(* CODESYS project devicelib.library
   Author: AMKO-Engineering
   Placeholder: Device_Library
   Title: Device_Library
   Version: 1.2.0.0
   Description: Device library of AMKO-Engineering.
   Company: AMKO-Engineering

Project tree, tasks and I/O mapping:
  libraries: System_Library, * (AMKO-Engineering); Tc2_MC2, 3.3.38.0 (Beckhoff Automation GmbH); Tc2_MC2_Drive, 3.3.21.0 (Beckhoff Automation GmbH); Tc2_Standard, 3.3.3.0 (Beckhoff Automation GmbH); Utilities_Library, * (AMKO-Engineering)
  Actuators/
    Cylinder/
      DataTypes/
        data type E_CylinderCmd
        data type E_ValveResetState
      Functions/
        function block Fb_DevCylWithFbk [ST]: ExecCalcTimers, ExecDirection, ExecSetFeedback, ExecTimeout, CmdSimulate, CmdTeach, Init
        function block FB_DevValve [ST]: ExecSetFeedback, ExecSetOutPuts, CmdClose, CmdHold, CmdManual, CmdOpen, CmdReset, CmdSafeStop, CmdTeach, Init
      MLTFunctions/
        function block Fb_DevSupportCyl [ST]: ExecCalc, ExecCylControl, ExecFaultHandling, Init_Support, Mod_ManualControl, Mod_SupportDown
  Axis/
    DataTypes/
      data type E_AxisCmd
      data type UDT_AxisData
      data type UDT_AxVal
    FunctionBlocks/
      function block FB_Axis [ST]: GearAsSlave, GearOutSlave, GearSlaveDyn, GetActVal, Hold, Home, Init, Jog, MoveAbs, MoveModulo, MoveRelative, MoveVeloFwd, MoveVeloRev, Reset, Stop
      function block Fb_AxisNew [ST]: CmdGearDynamic, CmdGearIn, CmdGearOut, CmdHalt, CmdHome, CmdJog, CmdLimitVelocity, CmdMoveAbs, CmdMoveModulo, CmdMoveRelative, CmdMoveVelocity, CmdReset, CmdSafeSpeed, CmdSafeStop, Init, ExecGearDynamic, ExecGearIn, ExecGearOut, ExecHalt, ExecHome, ExecJog, ExecMoveAbsolute, ExecMoveModulo, ExecMoveRelative, ExecMoveVelocity, ExecEnable, ExecReadStatus, ExecReset, ExecSafeFunctions, METH_ExecuteMotionFunctions, METH_ExecuteOrganizationFunctions
    Interface/
  BaseFunctions/
    function block FB_DevBase [ST]: CmdReset, CmdSafeStop
  Buttons/
    DataTypes/
    Functions/
      function block FB_DevHMIButton [ST]
      function block FB_DevPushButton [ST]
      function block FB_DevPushbuttonLight [ST]
  Encoders/
    DataTypes/
    FunctionBlocks/
      function block FB_EncoderBase [ST]: FastTask
      function block FB_EncoderInput [ST]: FastTask
  GroupHandlers/
    ManualControlHandler/
      function block FB_DevManualHandler [CFC]
  Heaters/
    function block FB_DevPWMGenerator [ST]: CalcCycle, ExecSetOutput, CmdOutputCycle, CmdOutputOff, CmdOutputOn
  Lights/
    DataTypes/
      data type E_LightState
    Functions/
      function block Fb_DevLight [ST]: Mod_SetOutput
  Outputs/
    DigitalOutputs/
      function block FB_DigitalOutput [ST]: ExecSetFeedback, ExecSetOutput, CmdOn
  Sensors/
    DigitalSensor/
      DataTypes/
        data type Udt_DigitalSensor
      FunctionBlocks/
        function block Fb_DevDigitalInput [ST]
        function block Fb_DevDigitalInputFunctions [ST]
    FootPedals/
      DataTypes/
        data type E_FootpedalPos
      FunctionBlocks/
        function block FB_EfkaEB301A_FootPedal [ST]: ACT_ConvertGreycode, ACT_CreateEdges
  Version/
    global variables Global_Version
*)

// Actuators/Cylinder/DataTypes/E_CylinderCmd
(* cylinder commands *)
TYPE E_CylinderCmd :
(
	Cyl_Idle 		:= 0,// Jog Cylinder command Referance 0 Idle (wait for command)
	Cyl_Init 		:= 1,// Jog Cylinder command Referance 1 initialize Cylinder
	Cyl_Enable 		:= 2,// Jog Cylinder command Referance 2 enable
	Cyl_Disable 	:= 3,// Jog Cylinder command Referance 3 disable
	Cyl_Reset 		:= 4,// Jog Cylinder command Referance 4 reset
	Cyl_Hold 		:= 5,// Jog Cylinder command Referance 5 hold
	Cyl_Teach 		:= 6,// Jog Cylinder command Referance 6 teach timeout settings
	Cyl_Calculate 	:= 7,// Jog Cylinder command Referance 7 calculate timeout settings from parameters
	Cyl_Expand 		:= 8,// Jog Cylinder command Referance 8 expand
	Cyl_Retract 	:= 9 // Jog Cylinder command Referance 9 retract
);
END_TYPE

// Actuators/Cylinder/DataTypes/E_ValveResetState
{attribute 'qualified_only'}
{attribute 'strict'}
TYPE E_ValveResetState :
(
	Res_Idle 		:= 0,
	Res_Closed		:= 1,
	Res_Open		:= 2
);
END_TYPE

// Axis/DataTypes/E_AxisCmd
(* axis command structure *)
TYPE E_AxisCmd :
(
	Ax_Idle 		:= 0,// Axis command Referance 0 Axis Idle
	Ax_Init 		:= 1,// Axis command Referance 1 Initialize axis
	Ax_Enable 		:= 2,// Axis command Referance 2 Enable
	Ax_Disable 		:= 3,// Axis command Referance 3 Disable
	Ax_Reset 		:= 4,// Axis command Referance 4 Reset
	Ax_Hold 		:= 5,// Axis command Referance 5 Hold
	Ax_Home 		:= 6,// Axis command Referance 6 Home
	Ax_JogFwd 		:= 7,// Axis command Referance 7 Jog Forward
	Ax_JogRev 		:= 8,// Axis command Referance 8 Jog Reverse
	Ax_MoveRelative := 9,// Axis command Referance 9 Move axis relative
	Ax_MoveAbs 		:= 10,// Axis command Referance 11 Move absolute reverse
	Ax_MoveModulo 	:= 11,// Axis command Referance 11 Move Module
	Ax_MoveVeloFwd 	:= 12,// Axis command Referance 12 Move velocity forward
	Ax_MoveVeloRev 	:= 13,// Axis command Referance 13 Move velocity reverse
	Ax_HardStop 	:= 14,// Axis command Referance 14 hard stop or emergency stop
	Ax_SoftStop 	:= 15,// Axis command Referance 15 soft stop after motion command
	Ax_GearSlave 	:= 16,// Axis command Referance 16 gear axis as slave
	Ax_GearSlaveDyn	:= 17,// Axis command Referance 17 gear axis as slave dynamic
	Ax_GearOutSlave := 18,// Axis command Referance 18 gear out from Master axis 
	Ax_Maintenance	:= 50 // Axis Command referance 50 maintenance mode, axis enabled with no command active
);
END_TYPE

// Axis/DataTypes/UDT_AxisData
TYPE UDT_AxisData:
STRUCT
	// ===== Axis name =====
		AxisName	: STRING 	; // Name of the axis (used for fault handling and identification)
		AxisNumber	: INT		; // Axis number 

	// ===== Fault data =====
		Message			: UDT_Fault 	; // Message data from Cylinder
		MessageActive	: BOOL			; // Message is active
		ErrorActive 	: BOOL 			;	// Axis in error state

	// ===== Axis Commands =====
		// ***** Enable command	*****
			CmdEnable		: BOOL 		; // Command enable axis
		// ***** Active commands *****
			AxisCmd			: E_AxisCmd ; // Axis command
			AxisSafeCmd		: E_AxisCmd	; // Axis safe command
			AxisAct			: E_AxisCmd ; // Axis Active status
		// ***** Command Modes *****
			CmdHomingMode 	: MC_HomingMode ; // Homing Mode ( MC_DefaultHoming, MC_Direct, MC_ForceCallibration, MC_ResetCallibration)
			CmdJogMode		: E_JogMode 	;
			CmdBuffermode	: MC_BufferMode	; // Buffermode used for command transition 	 
	// ===== Axis Safe commands =====
		SafeCmdLimitVelo: BOOL 	; // safe command limit velocity
		SafeCmdVelocity	: LREAL ; // Safe command velocity
		SafeCmdStop		: BOOL 	; // Stop command from safety or collision detection		
		SafeVeloLimit	: LREAL ; // safe velocity limit (link to FPAR)
	// ===== Status indication active =====
		ActHoming	: BOOL ; // Axis is homing
		ActBusy		: BOOL ; // Axis is Busy 
		ActMoving	: BOOL ; // Axis is moving
		ActAtVelo	: BOOL ; // Axis is at command velocity (only when written in Move velocity mode)

	// ===== Status indication done  =====
		FcoInit		: BOOL ; // Axis is initialised
		FcoIdle		: BOOL ; // Axis is idle enable required
		FcoEnabled	: BOOL ; // Axis is enabled
		FcoHomed	: BOOL ; // Axis is homed
		FcoGeared	: BOOL ; // Axis is geared to master axis
		FcoHeld		: BOOL ; // Axis is holding
		FcoStopped	: BOOL ; // Axis is stopped
		FcoReset	: BOOL ; // Axis reset done
		FcoReady 	: BOOL ; // Axis is ready for command
		FcoAtCmdPos	: BOOL ; // Axis is at command position (tol 0.2 deg)
		FcoCmdActive: BOOL ; // Axis new command values are active
		
	// ===== Move values =====
		Pos			: UDT_Axval	; // possition values (0 = infinite)
		Velocity 	: UDT_AxVal	; // Velocity values
		Accel		: UDT_Axval ; // Aceleration values
		Decel		: UDT_Axval ; // Deceleration values
		Torque		: UDT_Axval ; // Torque values
		EncTurnoverVal	: DINT 	; // Encoder turnover value
		TimeDisableDelay : TIME ; // Time off delay after axis move command (remove enable)
		
	// ===== Config Bits =====
		IcfCommandSpeedRpm	: BOOL ; // input speeds in Rpm
		IcfEnableForward 	: BOOL ; // Enable forward motion
 		IcfEnablereverse	: BOOL ; // Enable reverse motion
		IcfContinuous		: BOOL ; // continuous motion possible (no endpoint)
		IcfAlwaysEnable		: BOOL ; // 1 = Axis always enabled, 0 = Axis disabled at Idle 
		
	// ===== Master Axis =====
		MasterAxisRef	: REFERENCE TO AXIS_REF ; // Master axis reference (if applicable)
		GearMasterRev	: UINT	:= 1	; // Master Axis Gearing revolutions (Denominator)
		GearSlaveRev	: LREAL	:= 1	; // Slave Axis gearing revolutions (numerator)	
		ReverseSlave	: BOOL 	; // Reverse slave axis relative to master
		 
END_STRUCT
END_TYPE

// Axis/DataTypes/UDT_AxVal
TYPE UDT_AxVal :
STRUCT
	// ***** Velocity settings *****
		HardMax		: LREAL 	; // Hardware maximum set absolute maximum
		ManMax 		: LREAL		; // Manual maximum percentage of hardware max
		AutoMax		: LREAL		; // Automatic maximum percentage of hardware max
		HomeMax		: LREAL 	; // Homing maximum percentage of hardware max
		CmdVal		: LREAL 	; // Commanded value
		SafeVal		: LREAL		; // Command value after safety check
		PrevVal		: LREAL		; // previous command value 
		ActVal		: LREAL		; // Actual value
		ActModulo	: LREAL		; // [deg] Modulo position
		RefVal		: LREAL 	; // referance value (basic setting or home) 
END_STRUCT
END_TYPE

// Lights/DataTypes/E_LightState
(* discribes signal light state *)
TYPE E_LightState :
(
	Light_Off 		:= 0,// Jog Light state Referance 0 Light is off
	Light_BlinkSlow := 1,// Jog Light state Referance 1 Light blinking fast 
	Light_BlinkFast := 2,// Jog Light state Referance 2 light blinking slow
	Light_On 		:= 3 // Jog Light state Referance 3 Light permanently on
);
END_TYPE

// Sensors/DigitalSensor/DataTypes/Udt_DigitalSensor
TYPE Udt_DigitalSensor :
STRUCT
	Istatus		AT 	%I* : BOOL			;// Digital sensor, Direct input status
	ISensorEnable		: BOOL			;// Digital sensor, Input enable button
	tSensorDelay		: TIME 			;// Time before delayed signal becomes active 
	FcoSensorActive		: BOOL 			;// Digital sensor, Button active state
	FcoDelay			: BOOL			;// Digital sensor, Delayed input status (3 seconds) 
	FeStatus			: BOOL			;// Digital sensor, Falling edge of input signal	
	ReStatus			: BOOL			;// Digital sensor, Rising edge of input signal
	FcoFlipFlop			: BOOL			;// Digital sensor, feedback flip flop
	TetSensorActive		: TIME			;// Digital sensor, Time elapsed while button is active
END_STRUCT
END_TYPE

// Sensors/FootPedals/DataTypes/E_FootpedalPos
{attribute 'qualified_only'}
{attribute 'strict'}
TYPE E_FootpedalPos :
(
	eReverse2 	,
	eReverse1 	,
	eIdle		,
	eForward1	,
	eForward2	,
	eForward3	,
	eForward4	,
	eForward5	,
	eForward6	,
	eForward7	,
	eForward8	,
	eForward9	,
	eForward10	,
	eForward11	,
	eForward12	,
	eForward13	,
	eFalse			
) INT; 
END_TYPE

// Version/Global_Version
{attribute 'TcGenerated'}
{attribute 'no-analysis'}
{attribute 'linkalways'}
// This function has been automatically generated from the project information.
VAR_GLOBAL CONSTANT
	{attribute 'const_non_replaced'}
	stLibVersion_Device_Library : ST_LibVersion := (iMajor := 1, iMinor := 2, iBuild := 0, iRevision := 0, nFlags := 0, sVersion := '1.2.0.0');
END_VAR

// Actuators/Cylinder/Functions/Fb_DevCylWithFbk
FUNCTION_BLOCK PUBLIC Fb_DevCylWithFbk EXTENDS FB_DevValve
VAR_INPUT
	bIcfFbkOpenPresent 	: BOOL := FALSE ; // Feedback for cylinder open is present 
	bIcfFbkClosedPresent: BOOL := FALSE ; // Feedback for Cylinder closed is present
	bIcfTimeChecked		: BOOL := TRUE 	; // Cylinder timing is checked = default true
	nMargin				: LREAL:= 10	; // % of tollerance in move speed 
END_VAR
VAR_OUTPUT
	// ===== Teach function =======
	bCmdCopyTimeParam 	: BOOL	:= FALSE 	;// Cylinder, Command to higher level copy toucht time to parameters
	nOutTimeToClose		: LREAL	:= 0		; // Time it takes for valve to open	
	nOutTimeToOpen		: LREAL := 0		; // Time it takes for valve to close
	bFeClosed			: BOOL 	:= FALSE	; // closed sensor falling edge
	bReClosed			: BOOL 	:= FALSE	; // closed sensor rising edge
	bFeOpen				: BOOL 	:= FALSE 	; // Open sensor falling edge
	bReOpen				: BOOL 	:= false 	; // open sensor rising edge 
END_VAR
VAR	
	bFcoCalcDone	: BOOL := FALSE ; // Calculate timers done 
	
	stTimesClose	: Udt_TimerBandwith ; // Timer bandwith for cylinder close
	stTimesOpen		: Udt_TimerBandwith	; // Timer bandwitch for cylinder open 
	
	fbSensorClosed	: Fb_DevDigitalInputFunctions ; // Digital sensor function closed detection
	fbSensorOpen	: Fb_DevDigitalInputFunctions ; // Digital sensor function open detection
	
	fbTimerOpen		: TON ; // Timer for cylinder to open
	fbTimerClose 	: TON ; // Timer for cylinder to close
	fbTimerTeach	: TON ; // timer for teachin cylinder 

	rtCmdWriteParam	: R_TRIG ; // Write parameter rising edge trigger 
	// Simulation
	fbTimerSimOpen 	: TON 	; 
	fbTimerSimClose	: TON 	; 
	
	// Time Cylinder valid 
	bTriggerTimeClose	: BOOL ;
	bTriggerTimeOpen	: BOOL ;

END_VAR

IF NOT bInitOk THEN
	RETURN;
ELSE
	SUPER^();
END_IF 

// ====== Check direction of movement =======
	ExecDirection();
	
// ====== Check movement speed =======
	IF bFcoCalcDone AND bIcfTimeChecked THEN 
		ExecTimeout();
	END_IF
	
// ====== Calculate timers =======
	IF nTimeToCloseMs <> stTimesClose.Nominal OR nTimeToOpenMs <> stTimesOpen.Nominal OR NOT bFcoCalcDone THEN 
		bFcoCalcDone := FALSE ;
		ExecCalcTimers();
	END_IF

// ==== set timer output feedback 
	nOutTimeToClose := stTimesClose.Nominal ;
	nOutTimeToOpen	:= stTimesOpen.Nominal	;	

// ===== send write parameters command ======	
	rtCmdWriteParam(CLK := bFcoCalcDone);
	bCmdCopyTimeParam := rtCmdWriteParam.Q	;

METHOD PRIVATE ExecCalcTimers : BOOL
VAR
END_VAR
// ====== Calculate close times ======
	stTimesClose.Nominal 	:= nTimeToCloseMs ;
	stTimesClose.Maximum 	:= nTimeToCloseMs * (1 + (nMargin / 100));
	stTimesClose.Minimal 	:= nTimeToCloseMs * (1 - (nMargin / 100));

// ====== Calculate open times ======
	stTimesOpen.Nominal 	:= nTimeToOpenMs ;
	stTimesOpen.Maximum 	:= nTimeToOpenMs * (1 + (nMargin / 100));
	stTimesOpen.Minimal 	:= nTimeToOpenMs * (1 - (nMargin / 100));
	
// ====== Set feedback =======
	bFcoCalcDone := TRUE ;
END_METHOD

METHOD PRIVATE ExecDirection : BOOL
VAR_INPUT
END_VAR
// ===== Check direction commands =====
 	IF q_Close AND fbSensorOpen.bReStatus AND NOT q_Open THEN
		stFault.MessageNumber	:= E_MessageNumbers.CF_WrongDirection 	;
		stFault.Discription		:= 'Cylinder Opening instead of closing';
		stFault.FaultType		:= E_FaultTypes.CF 					;
		bErrorActive			:= TRUE 								;
		refFbFault.CmdAddFault( stFault );
	ELSIF q_Open AND fbSensorClosed.bReStatus AND NOT q_close THEN
		stFault.MessageNumber	:= E_MessageNumbers.CF_WrongDirection 	;
		stFault.Discription		:= 'Cylinder closing instead of opening';
		stFault.FaultType		:= E_FaultTypes.CF 					;
		bErrorActive			:= TRUE 								;
		refFbFault.CmdAddFault( stFault );
	END_IF
END_METHOD

METHOD PROTECTED ExecSetFeedback : BOOL
VAR_INPUT
END_VAR
// ====== Call sensor Open function =======
	IF bIcfFbkClosedPresent THEN 
		fbSensorClosed();
		bFco_Closed := fbSensorClosed.bFcoInputActive ;
		bFeClosed 	:= fbSensorClosed.bFeStatus ;
		bReClosed 	:= fbSensorClosed.bReStatus ;
	ELSE 
		fbTOnClose	(IN 	:= q_Close, PT 	:= LREAL_TO_TIME(nTimeToCloseMs))	;
		bFco_Closed := fbTOnClose.Q ;
	END_IF

// ====== Call sensor Close function =======
	IF bIcfFbkOpenPresent THEN 
		fbSensorOpen() 	;
		bFco_open 	:= fbSensorOpen.bFcoInputActive ;
		bFeOpen		:= fbSensorOpen.bFeStatus;
		bReOpen		:= fbSensorOpen.bReStatus;
	ELSE 
		FbTOnOpen	(IN 	:= q_Open, PT 	:= LREAL_TO_TIME(nTimeToOpenMs))	;
		bFco_Open := FbTOnOpen.Q ;
	END_IF

// ====== set outputs =======
	bReady		:= bFco_Closed OR bFco_Open ;
END_METHOD

METHOD PRIVATE ExecTimeout : BOOL
VAR_INPUT
END_VAR
VAR
	nTimePassedMs : LREAL ;
END_VAR
// ====== Set triggers ======
	IF q_Close  AND bFco_Open THEN 
		bTriggerTimeClose := TRUE ;
	ELSIF q_Open OR bFco_Closed  THEN 
		bTriggerTimeClose := FALSE ;
	END_IF

	IF q_Open  AND bFco_Closed THEN 
		bTriggerTimeOpen := TRUE ;
	ELSIF q_Close OR bFco_Open THEN
		bTriggerTimeOpen := FALSE ;
	END_IF
	
//======= run timers =======
	IF bIcfFbkClosedPresent THEN 
		fbTimerClose(IN := q_Close, PT := T#1M);
	END_IF	
	
	IF bIcfFbkOpenPresent THEN 
		fbTimerOpen	(IN := q_Open , PT := T#1M);
	END_IF

//====== Run timeout checks for cylinder close =======
	nTimePassedMs:= TIME_TO_LREAL(fbTimerClose.ET);
	
	IF bIcfFbkClosedPresent THEN 
		IF bTriggerTimeClose THEN 
			IF fbSensorClosed.bReStatus THEN 
				IF nTimePassedMs < stTimesClose.Minimal THEN 
					// send message to HMI 
					stFault.MessageNumber	:= E_MessageNumbers.CF_MoveToFast 	;
					stFault.Discription		:= 'Cylinder closing to fast'		;
					stFault.FaultType		:= E_FaultTypes.CF 				;
					bErrorActive			:= TRUE 							;
					refFbFault.CmdAddFault( stFault );
				ELSIF	nTimePassedMs > stTimesClose.Maximum  THEN
					// send message to HMI 
					stFault.MessageNumber	:= E_MessageNumbers.CF_MoveToSlow 	;
					stFault.Discription		:= 'Cylinder closing to Slow'		;
					stFault.FaultType		:= E_FaultTypes.CF 				;
					bErrorActive			:= TRUE 							;
					refFbFault.CmdAddFault( stFault );
				END_IF
			END_IF
		END_IF
	END_IF	

//====== Run timeout checks for cylinder Open =======
	nTimePassedMs:= TIME_TO_REAL(fbTimerOpen.ET);

	IF bIcfFbkOpenPresent THEN 
		IF bTriggerTimeOpen THEN 
			IF fbSensorOpen.bReStatus THEN 
				IF nTimePassedMs < stTimesOpen.Minimal THEN 
					// send message to HMI 
					stFault.MessageNumber	:= E_MessageNumbers.CF_MoveToFast 	;
					stFault.Discription		:= 'Cylinder Opening to fast'		;
					stFault.FaultType		:= E_FaultTypes.CF 				;
					bErrorActive			:= TRUE 							;
					refFbFault.CmdAddFault( stFault );
				ELSIF	nTimePassedMs > stTimesOpen.Maximum  THEN
					// send message to HMI 
					stFault.MessageNumber	:= E_MessageNumbers.CF_MoveToSlow 	;
					stFault.Discription		:= 'Cylinder Opening to Slow'		;
					stFault.FaultType		:= E_FaultTypes.CF 				;
					bErrorActive			:= TRUE 							;
					refFbFault.CmdAddFault( stFault );
				END_IF
			END_IF
		END_IF
	END_IF
END_METHOD

METHOD PUBLIC CmdSimulate : BOOL
VAR_INPUT
	bFbkReverse		: BOOL := FALSE ; 
	tTimeSimOpen	: TIME := T#1S 	;
	tTimeSimClose	: TIME := T#1S 	;  
END_VAR
VAR
	bCmdSimulate : BOOL := TRUE ;
END_VAR
// Run timers when cylinder is active 
	fbTimerSimOpen	(IN := q_Open	, PT := tTimeSimOpen);
	fbTimerSimClose	(IN := q_Close	, PT := tTimeSimClose);

 // set feedback sensors to simulate
	fbSensorOpen.bCmdSimulate 	:= TRUE ;
	fbSensorClosed.bCmdSimulate := TRUE ;

 // set simulated feedback state 
	IF bFbkReverse THEN 
		fbSensorClosed.bSimState:= fbTimerSimOpen.Q 	;
		fbSensorOpen.bSimState	:= fbTimerSimClose.Q 	; 	
	ELSE 
		fbSensorClosed.bSimState:= fbTimerSimClose.Q 	;
		fbSensorOpen.bSimState	:= fbTimerSimOpen.Q 	; 	
	END_IF
END_METHOD

METHOD PUBLIC CmdTeach : BOOL
VAR_INPUT
END_VAR
// ====== turn off time check function until new calculation cycle =======
	bFcoCalcDone := false ;

// ====== teach cylinder from hardware inputs ======
	fbTimerTeach	(PT:= T#60S);
	fbTimerSwitchDir(PT:= T#1S); 
// ====== time cylinder cycles ======
	// ===== Start test loop =====
	IF bFco_Closed AND fbTimerSwitchDir.Q THEN
		bCmdClose 			:= FALSE;
		bCmdOpen 			:= TRUE ;
		fbTimerSwitchDir.IN	:= FALSE; 
		fbTimerTeach.IN 	:= TRUE ;
	ELSIF bFco_Open AND fbTimerSwitchDir.Q THEN
		bCmdClose 			:= TRUE ;
		bCmdOpen 			:= FALSE;
		fbTimerSwitchDir.IN	:= FALSE; 
		fbTimerTeach.IN 	:= TRUE ;
	ELSIF NOT bCmdClose AND NOT bCmdOpen THEN 
		bCmdClose 			:= TRUE ;
		bCmdOpen 			:= FALSE;
		fbTimerTeach.IN 	:= TRUE ;
	END_IF

// ====== start timing ========
	IF bCmdClose AND bFco_Closed THEN 
		IF fbTimerTeach.IN THEN
			nTimeToCloseMs 	:= TIME_TO_LREAL(fbTimerTeach.ET);
		END_IF
		fbTimerSwitchDir.IN := TRUE 		;
		fbTimerTeach.IN 	:= FALSE 		;
	ELSIF bCmdOpen AND bFco_Open THEN 
		IF fbTimerTeach.IN THEN
			nTimeToOpenMs		:= TIME_TO_LREAL(fbTimerTeach.ET);
		END_IF
		fbTimerSwitchDir.IN := TRUE 		;
		fbTimerTeach.IN 	:= FALSE 		;
	END_IF
END_METHOD

METHOD PUBLIC Init : BOOL
VAR_INPUT
	// Valve data
	nInValveNumber	: UDINT				:= 0		; // Cylinder identification number
	// Command state
	eResetState		: E_ValveResetState := 0		; // Cylinder reset state variable (default is idle) 
	eSafeState		: E_ValveResetState	:= 0		; // Valve safe state
END_VAR
bFcoCalcDone := FALSE;

// Enable sensor feedback
fbSensorClosed.bEnable	:= TRUE ;
fbSensorOpen.bEnable	:= TRUE ;

// Call feedback sensors 
ExecSetFeedback(); 

SUPER^.Init(nInValveNumber, eResetState, eSafeState);
END_METHOD

END_FUNCTION_BLOCK

// Actuators/Cylinder/Functions/FB_DevValve
FUNCTION_BLOCK PUBLIC FB_DevValve EXTENDS FB_DevBase
VAR_INPUT
	// Timer values
	nTimeToCloseMs	: LREAL			:= 50		; // Time it takes for valve to open	
	nTimeToOpenMs	: LREAL			:= 50		; // Time it takes for valve to close
END_VAR
VAR_OUTPUT
	// ===== Status indicators =======
		bFco_Closed		:	BOOL := FALSE ;
		bFco_Open		: 	BOOL := FALSE ;
END_VAR
VAR
	// Hardware links 
		q_Open			AT %Q* : BOOL := FALSE 	; // Open valve
		q_Close 		AT %Q* : BOOL := FALSE	; // Close valve
	// Internal commands
		bCmdClose 	: BOOL := FALSE ; // close valve 
		bCmdOpen	: BOOL := FALSE ; // Open valve
		bCmdHold	: BOOL := FALSE ; // Hold valve status change
	// Time functions 
		fbTOnClose	: TON	; // Timer for valve close
		FbTOnOpen	: TON 	; // Timer for valve Open
		fbTimerSwitchDir: TON ; // Time for teach function switch direction 
	// reset and safe state
		eResetState		: E_ValveResetState := 0		; // Cylinder reset state variable (default is idle) 
		eSafeState		: E_ValveResetState	:= 0		; // Valve safe state
END_VAR

// ===== hold all actions if not initialized ======
IF NOT bInitOk THEN
	RETURN;
ELSE
	SUPER^();
END_IF 


// ====== Set Outputs =======
	ExecSetOutPuts();

// ===== collect feedback ======
	ExecSetFeedback();

// ===== Message test function ======
	IF bMessageTest THEN 
		stFault.Active 			:= TRUE ;
		stFault.Discription 	:= 'This is a test message from fb_DevValve';
		stFault.MessageNumber 	:= E_MessageNumbers.OM_MessageTest ;
		stFault.FaultType		:= Utilities_Library.E_FaultTypes.OM ;
		refFbFault.CmdAddFault( stFault );
	END_IF

METHOD PROTECTED ExecSetFeedback : BOOL
VAR_INPUT
END_VAR
// ====== Set timers =======
	fbTOnClose	(PT 	:= LREAL_TO_TIME(nTimeToCloseMs))	;
	FbTOnOpen	(PT		:= LREAL_TO_TIME(nTimeToOpenMs))	;

// ====== Set timed feedback ======
	IF q_Close THEN 
		fbTOnClose.IN 	:= TRUE ;
		fbTOnopen.IN 	:= FALSE;
	ELSIF q_Open THEN 
		fbTOnClose.IN 	:= FALSE;
		FbTOnOpen.IN	:= TRUE ;
	ELSE 
		fbTOnClose.IN 	:= FALSE;
		FbTOnOpen.IN	:= FALSE;
	END_IF
	
// ====== set outputs =======
	bFco_Closed := fbTOnClose.Q ;
	bFco_Open	:= FbTOnOpen.Q	;
	bReady		:= bFco_Closed OR bFco_Open ;
END_METHOD

METHOD PROTECTED ExecSetOutPuts : BOOL
VAR_INPUT
END_VAR
// ======= Set Outputs according to commands and check safety features =======
	IF bEnable	OR bCmdManual THEN  
		IF NOT bCmdHold THEN 
			q_Close	:= bCmdClose;
			q_Open	:= bCmdOpen	;
		END_IF
	ELSE
		CASE eSafeState OF 
			E_ValveResetState.Res_Idle:
				q_Close	:= bFco_Closed;		
				q_Open 	:= bFco_Open;
			E_ValveResetState.Res_Closed:
				q_Close	:= TRUE	;		
				q_Open 	:= FALSE;
			E_ValveResetState.Res_Open:
				q_Close	:= FALSE;		
				q_Open 	:= TRUE	;
		END_CASE
		bCmdClose 	:= bFco_Closed 	;
		bCmdOpen	:= bFco_Open	;
		bCmdHold	:= FALSE ; 
	END_IF
END_METHOD

METHOD PUBLIC CmdClose : BOOL // close valve or retract cylinder
VAR_INPUT
END_VAR
// ====== Set close command if enabled ======
	bCmdClose 	:= TRUE	;		
	bCmdOpen 	:= FALSE;
	
// ===== Set feedback ======
	CmdClose := bFco_Closed ;
END_METHOD

METHOD PUBLIC CmdHold : BOOL
VAR_INPUT
END_VAR
// ====== set hold command =====
	bCmdHold := TRUE ;
END_METHOD

METHOD PUBLIC CmdManual : BOOL
VAR_INPUT
	bCmdOpen	: BOOL ; // open valve 
	bCmdClose	: BOOL ; // Close valve
	bCmdTeach	: BOOL ; // Teach valve  
END_VAR
// Enable manual commands
bCmdManual S= TRUE ;

// execute manual command 
	IF bCmdOpen THEN 
		CmdOpen();
	ELSIF bCmdClose THEN 
	 	CmdClose(); 
	ELSIF bCmdTeach THEN
		CmdTeach ();
	END_IF
END_METHOD

METHOD PUBLIC CmdOpen : BOOL // Open valve or retract cylinder
VAR_INPUT
END_VAR
// ====== Set open command if enabled ======
	bCmdClose 	:= FALSE;		
	bCmdOpen 	:= TRUE	;
	
// ===== Set feedback ======
	CmdOpen := bFco_Open ;
END_METHOD

METHOD CmdReset : BOOL
VAR_INPUT
END_VAR
// ====== Set outputs according to reset state =======
	IF bEnable THEN 
		CASE eResetState OF 
			E_ValveResetState.Res_Idle:
				bCmdClose 	:= FALSE;		
				bCmdOpen 	:= FALSE;
			E_ValveResetState.Res_Closed:
				bCmdClose 	:= TRUE	;		
				bCmdOpen 	:= FALSE;
			E_ValveResetState.Res_Open:
				bCmdClose 	:= FALSE;		
				bCmdOpen 	:= TRUE	;
		ELSE
			;
		END_CASE
	END_IF
// ======= Reset Error bit ======
	bErrorActive 	:= FALSE;
	bBussy			:= FALSE;
END_METHOD

METHOD PUBLIC CmdSafeStop : BOOL
VAR_INPUT
END_VAR
CASE eSafeState OF 
	E_ValveResetState.Res_Idle:
		bDevIsSafe := bFco_Closed OR bFco_Open ;
	E_ValveResetState.Res_Closed:
		bDevIsSafe := bFco_Closed ;
	E_ValveResetState.Res_Open:
		bDevIsSafe := bFco_Open ;
END_CASE

CmdSafeStop := bDevIsSafe ;
END_METHOD

METHOD PUBLIC CmdTeach : BOOL
VAR_INPUT
END_VAR
// ====== teach cylinder from hardware inputs ======
	fbTimerSwitchDir(PT:= T#1S); 
// ===== Start test loop =====
IF bFco_Closed AND fbTimerSwitchDir.Q THEN
	bCmdClose 			:= FALSE;
	bCmdOpen 			:= TRUE ;
	fbTimerSwitchDir.IN	:= FALSE; 
ELSIF bFco_Open AND fbTimerSwitchDir.Q THEN
	bCmdClose 			:= TRUE ;
	bCmdOpen 			:= FALSE;
	fbTimerSwitchDir.IN	:= FALSE; 
ELSIF NOT bCmdClose AND NOT bCmdOpen THEN 
	bCmdClose 			:= TRUE ;
	bCmdOpen 			:= FALSE;
END_IF
END_METHOD

METHOD PUBLIC Init : BOOL
VAR_INPUT
	// Valve data 
	nInValveNumber	: UDINT				:= 0		; // Cylinder identification number
	// Command state
	eResetState		: E_ValveResetState := 0		; // Cylinder reset state variable (default is idle) 
	eSafeState		: E_ValveResetState	:= 0		; // Valve safe state
END_VAR
// ====== Set message information =======
//	refFbMessage 			:= GVL_Message.fbDefaultMessageArray;
	stFault.ComponentType	:= E_ComponentTypes.Cylinder 		;
	stFault.LocationName	:= F_FBNameFromPath(sPath := sPath)	;	
	stFault.LocationNumber:= nInValveNumber 					;
	
// ====== Set outputs according to reset state =======
	THIS^.eResetState 	:= eResetState 	;
	THIS^.eSafeState	:= eSafeState	;	

	IF bEnable THEN 
		CASE eResetState OF 
			E_ValveResetState.Res_Idle:
				bCmdClose 	:= bFco_Closed	;		
				bCmdOpen 	:= bFco_Open	;
			E_ValveResetState.Res_Closed:
				bCmdClose 	:= TRUE;		
				bCmdOpen 	:= FALSE;
			E_ValveResetState.Res_Open:
				bCmdClose 	:= FALSE;		
				bCmdOpen 	:= TRUE ;
		END_CASE
	END_IF
// ======= Reset Error bit ======
	bErrorActive 	:= FALSE;
	bBussy			:= FALSE;
	
// ====== Set init status bit =======
	bInitOk := TRUE ;
END_METHOD

END_FUNCTION_BLOCK

// BaseFunctions/FB_DevBase
{attribute 'reflection'}
FUNCTION_BLOCK PUBLIC FB_DevBase
VAR_INPUT
	nModuleId		: UDINT 			:= 	1 		; // Higher level module ID
	bEnable			: REFERENCE TO BOOL := GVL_Main.stModules[nModuleId].bEnabled	; // Module enable signal reference
	bReset 			: REFERENCE TO BOOL := GVL_Main.stModules[nModuleId].bResetting ; // reset command bit reference (default = Module[id].bresetting)
	refFbFault		: REFERENCE TO Fb_FaultHandler 	:= GVL_Main.stModules[nModuleId].fbFaultHandler ; // reference to fault handler ( default = Module[id].FbFaulthandler)
END_VAR
VAR_OUTPUT
	sDevActiveState	: STRING 		:= 'Idle'	; // active state of device 
	bInitOk			: BOOL 			:= FALSE 	; // function is initialized
	bBussy 			: BOOL 			:= FALSE 	; // device is busy
	bReady			: BOOL 			:= FALSE 	; // device is ready for new command 
	bDevIsSafe		: BOOL 			:= FALSE	; // Device is locked and safe
	bErrorActive	: BOOL			:= FALSE	; // device Error active 
END_VAR
VAR
	// Feedback request
	bMessageTest	: BOOL  		:= FALSE	; // Send test message from device
	// ===== Fault data =====
	stFault			: UDT_Fault	; // Fault data from device
	// internal commands 
	bCmdManual 		: BOOL		; // enable manual control functions (thus disable automatic)
	// Function path 
	{attribute 'instance-path'} 
    {attribute 'noinit'}
	sPath			: STRING	; // Path name of function (used for manual reference)
	sDevName		: STRING 	; // Name of device distilled from the path 
END_VAR

// Get device name from function
IF sDevName = '' THEN 
	sDevName := F_FBNameFromPath(sPath := sPath);
END_IF
// Call reset function 
IF bReset THEN 
	CmdReset();
END_IF

METHOD CmdReset : BOOL
VAR_INPUT
END_VAR
END_METHOD

METHOD PUBLIC CmdSafeStop : BOOL
VAR_INPUT
END_VAR
// check if device is safe
bDevIsSafe 	:= bInitOk AND NOT bEnable ;
CmdSafeStop := bDevIsSafe ;
END_METHOD

END_FUNCTION_BLOCK

// Sensors/DigitalSensor/FunctionBlocks/Fb_DevDigitalInputFunctions
FUNCTION_BLOCK PUBLIC Fb_DevDigitalInputFunctions EXTENDS Fb_DevDigitalInput
VAR_OUTPUT
	bFcoDelay			: BOOL			;// Digital sensor, Delayed input status (3 seconds) 
	bFeStatus			: BOOL			;// Digital sensor, Falling edge of input signal	
	bReStatus			: BOOL			;// Digital sensor, Rising edge of input signal
	bFcoFlipFlop		: BOOL			;// Digital sensor, feedback flip flop
	TetInputActive		: TIME			;// Digital sensor, Time elapsed while button is active
END_VAR
VAR
	// ***** Fucntion blocks *****
		FB_delIStatus: TON; // Timer function for delayed input status 
		FB_feIStatus: F_TRIG; // generate falling edge pulse edge from Istatus
		FB_reIStatus: R_TRIG; // generate falling edge pulse edge from Istatus
		FB_rsIStatus: RS; // Set Reset function for flip flop input
END_VAR

SUPER^();

// ====== process functions if enabled ======
	// ***** Set Delayed inputs and time elapsed ****
		FB_delIStatus(	IN:= bFcoInputActive,
						PT:= tDelay , 
						Q=> bFcoDelay , 
						ET=> TetInputActive 
					  ); // Generate delayed input status from push button input status
	// ***** Edge triggers *****
		FB_feIStatus(CLK:= bFcoInputActive , Q=> bFeStatus ); // generate falling edge pulse on pushbutton input
		FB_reIStatus (Clk := bFcoInputActive , Q => bReStatus); // Generate rising edge from push button input signal
	// ***** Flip Flop *****
		FB_rsIStatus(	SET:= bFeStatus AND NOT bFcoFlipFlop , 
						RESET1:= bFeStatus AND bFcoFlipFlop , 
						Q1=> bFcoFlipFlop 
					 ); // Generate set reset function from pushbutton input status

END_FUNCTION_BLOCK

// Sensors/DigitalSensor/FunctionBlocks/Fb_DevDigitalInput
FUNCTION_BLOCK PUBLIC Fb_DevDigitalInput 
VAR_INPUT
	bEnable			: BOOL  := TRUE ; // Enable input functions
	tDelay			: TIME 	:= T#1S	;// Time before delayed signal becomes active 
	bCmdSimulate	: BOOL 	:= FALSE ;// Simulate sensor Input 
	bSimState		: BOOL 	:= FALSE ;// Simulated sensor state
END_VAR
VAR_OUTPUT
	bFcoInputActive		: BOOL 			;// Digital sensor, Button active state
END_VAR
VAR
	Istatus		AT 	%I* : BOOL			;// Digital sensor, Direct input status
END_VAR

// ***** Direct input when enabled *****
IF bEnable THEN 
	IF bCmdSimulate  THEN 
		bFcoInputActive := bSimState ;
		bCmdSimulate	:= FALSE ;  
	ELSE
		bFcoInputActive := Istatus ;
	END_IF
ELSE 
	bFcoInputActive := FALSE ;
END_IF

// ***** Simulate sensor ******

END_FUNCTION_BLOCK

// Actuators/Cylinder/MLTFunctions/Fb_DevSupportCyl
FUNCTION_BLOCK PUBLIC Fb_DevSupportCyl EXTENDS Fb_DevCylWithFbk
VAR_INPUT
	// Traverse data
	stTraverseAxisRef	: AXIS_REF 			; // Axis reference
	nHandCartPos		: LREAL 			; // Position of hand cart
	tMindownTime		: TIME	:= T#1S		; // minimum time down before it can go up again 
END_VAR
VAR_OUTPUT
	bStopAll			: BOOL := TRUE 	; // Support fault stop all motions 
	// feedback 
	bSupportOk			: BOOL := FALSE 	; // Support is running ok
	 
END_VAR
VAR
	bCmdSupportDown		: BOOL 	:= FALSE 	; // External command to move support down 
	// Support data
	nSupportPosition	: LREAL := 0 		; // possition of support cylinder in reference to the home position 
	nSupportWidth		: LREAL := 100		; // width of support cylinder 
	// Traverse data 
	nTravMaxAcc				: LREAL ; // traverse maximum acceleration 
	nTravMaxDec				: LREAL ; // traverse maximum deceleration 
	nTraverseLength			: LREAL	:= 550		; // Length of sewing head Traverse 
	nTraverseFlagPosition	: LREAL	:= 0		; // position of flag in reference to edge of Traverse 
	
	// handcart data
	nHandCartLength			: LREAL := 100	; // Length of hand cart 
	nHandCartClearance		: LREAL := 300	; // Clearance around cart in which support is down
	
	// safety values 	
	nMinSafeDistanceDown: LREAL := 200	; // Minimum distance for support to move down

	// Traverse triggers 
	nMinStopDistance 	: 	LREAL 	:= 10		; // Minimum stopping distance required[mm]
	nTriggerDown		: 	LREAL	:= 100		; // trigger distance for support to go down[mm]
	nTriggerUp			: 	LREAL	:= 50 		; // trigger distance for support to move up[mm]
	nTriggerPosDownFw	:	LREAL 	; // trigger position for support to move down when moving forward [mm]
	nTriggerPosCheckDownFw: LREAL 	; // trigger for safety check is cylinder is down when mocing forward [mm]
	nTriggerPosDownRe	: 	LREAL 	; // trigger position for support to move down when moving reverse [mm]
	nTriggerPosCheckDownRe: LREAL 	; // trigger for safety check is cylinder is down when mocing reverse [mm]

	nTriggerPosUpFw		: 	LREAL	; // Trigger position for support to move Up [mm]
	nTriggerPosUprev	: 	LREAL	; // Trigger position for support to move Up [mm]
	
	// handcart down positions
	nCartCmdDownHigh	: LREAL ; // hand cart position for cylinder to go down high limit
	nCartCmdDownLow		: LREAL ; // hand cart Position for cylinder to go down low limit 
	
	fbTimerStartup		:	TON		; // Startup time before support down check
	
	// Support down trigger
	bSupportClose 	: BOOL 	; // Support close command
	tonSupportDown 	: TON 	; // support Down command
	
END_VAR

IF NOT bInitOk THEN
	bStopAll	:= TRUE ; 
	RETURN;
ELSE
	;
END_IF 

// ======= Enable/ disable support cylinder dependent functions =======
	bStopAll := bErrorActive OR bCmdManual OR NOT bEnable ; 	

// ======= Activate cylinder ======	
SUPER^();

// ====== Manual functions =====
	IF bCmdManual THEN 
		bCmdManual		:= FALSE ;	
		RETURN;
	END_IF
	
// ======= Calculate variables =======
	ExecCalc();	

// ======= Support cylinder control =======
	IF bCmdSupportDown THEN 
		CmdClose();
		IF bFco_Closed THEN 
			bCmdSupportDown := FALSE ;
		END_IF
 	ELSE
		ExecCylControl();
	END_IF

METHOD PROTECTED ExecCalc : BOOL
VAR_INPUT
END_VAR
VAR 
	nTriggerOffset 	: LREAL ;
	nMaxAccelDist	: LREAL ;
	nMaxVelocity	: LREAL ;
	nDecelDist		: LREAL	;
	nTraverseFront		: LREAL ; // front of Traverse distance from sensor flag
END_VAR
// ***** Calculate hardstop distance *****
	nMinStopDistance	:= (ABS(stTraverseAxisRef.NcToPlc.ActVelo) / 2) * (ABS(stTraverseAxisRef.NcToPlc.ActVelo) / nTravMaxDec);
	
// ***** Calculate speed dependant trigger offset *****
	nTriggerOffset := F_TriggerPosOffset( Velocity := ABS(stTraverseAxisRef.NcToPlc.ActVelo), nMoveTimeMs := stTimesClose.Maximum);

// ***** Calculate triggerdistance down *****
	nTriggerDown := (nSupportWidth / 2) + nMinStopDistance + nTriggerOffset;
	IF nTriggerDown < nMinSafeDistanceDown THEN 
		nTriggerDown := nMinSafeDistanceDown ;
	END_IF
	
// ***** Calculate triggerdistance Up *****
	nMaxAccelDist 	:= F_AccDecDistanceFromTime	(nAccelDecel:= nTravMaxAcc, nTimeMs := stTimesClose.Maximum);
	nMaxVelocity	:= F_TopVelocityFromTime	(nAccel 	:= nTravMaxAcc, nTimeMs := stTimesClose.Maximum);
	nDecelDist		:= F_AccDecDistanceFromVelo (nAccDecc	:= nTravMaxDec, nVelocity := nMaxVelocity);
	
	nTriggerUp	:= ((nSupportWidth / 2) + nMaxAccelDist + nDecelDist)* 1.1; // 1.1 is a %10 safety margint to account for cycle time 


// ***** calculate traverse lenght from sensor *****
	nTraverseFront := nTraverseLength - nTraverseFlagPosition ;

	
// ===== Calculate trigger positions =====
	// ***** positive direction positions *****
		nTriggerPosDownFw		:= nSupportPosition - nTriggerDown - nTraverseFront ;
		nTriggerPosCheckDownFw	:= nSupportPosition - (nSupportWidth / 2) - nTraverseFront - nMinStopDistance ; 
		nTriggerPosUpFw			:= nSupportPosition + nTraverseFlagPosition + nTriggerUp;
		
	// ***** negative direction positions *****
		nTriggerPosDownRe 		:= nSupportPosition + nTriggerDown + nTraverseFlagPosition ;
		nTriggerPosCheckDownRe	:= nSupportPosition + (nSupportWidth / 2) + nTraverseFlagPosition + nMinStopDistance; 
		nTriggerPosUprev		:= nSupportPosition - nTraverseFront - nTriggerUp;
	
// ===== calculate hand cart trigger positions ======
	nCartCmdDownHigh 	:= nSupportPosition + nHandCartClearance ;
	nCartCmdDownLow		:= nSupportPosition - nHandCartClearance - nHandCartLength  ;
END_METHOD

METHOD PROTECTED ExecCylControl : BOOL
VAR
	nTravPos : LREAL ;
END_VAR
// ===== copy position in temporary var (for readability ) ======
	nTravPos := stTraverseAxisRef.NcToPlc.ActPos ; 

// ===== Trigger Support cylinder =====
	IF nHandCartPos >= nCartCmdDownLow AND nHandCartPos <= nCartCmdDownHigh THEN  
		bSupportClose := TRUE ;
	ELSIF 	stTraverseAxisRef.Status.PositiveDirection 
		AND	nTravPos >= nTriggerPosDownFw 
		AND nTravPos <= nTriggerPosUpFw 
		THEN 
		bSupportClose := TRUE ;
	ELSIF 	stTraverseAxisRef.Status.NegativeDirection  
		AND nTravPos <= nTriggerPosDownRe 
		AND nTravPos >= nTriggerPosUprev 
		THEN 
		bSupportClose := TRUE ;
	ELSIF	nTravPos > nTriggerPosUprev AND nTravPos < nTriggerPosUpFw THEN 
		bSupportClose := TRUE ;
	ELSE
		bSupportClose := FALSE ;
	END_IF

// ===== Run filter timer =====
	tonSupportDown(IN := bFco_Closed, PT := tMindownTime);	

// ===== Set Cylinder command ======
	IF bSupportClose THEN 
		CmdClose() ;
	ELSIF tonSupportDown.Q THEN 
		CmdOpen();
	END_IF
END_METHOD

METHOD PROTECTED ExecFaultHandling : BOOL
VAR
	bEnableCheck: BOOL ; // enable check functions 
	nActPos		: LREAL; // actual position of traverse axis (for readability)	 
	bActMovFwd	: BOOL ; // traverse is moving in positive direction
	bActMovRev	: BOOL ; // traverse is moving in negative direction
END_VAR
// ====== Write axis position to temporary variable to improver readability =======
	nActPos := stTraverseAxisRef.NcToPlc.ActPos ;
	IF stTraverseAxisRef.Status.Moving THEN 
		bActMovFwd := stTraverseAxisRef.Status.PositiveDirection ; 
		bActMovRev := stTraverseAxisRef.Status.NegativeDirection ; 
	ELSE
		bActMovFwd := FALSE ; 
		bActMovRev := FALSE ; 
	END_IF
	
// ====== Alway check if cylinder is down when within minimum range ======
	fbTimerStartup(IN := NOT bErrorActive, PT := LREAL_TO_TIME(nTimeToCloseMs));
	
	IF fbTimerStartup.Q 
	AND	nActPos > nTriggerPosUprev 
	AND nActPos < nTriggerPosUpFw 
	AND NOT fbSensorClosed.bFcoInputActive  THEN 	
		// Set error to active (stop traverse axis) 
		bErrorActive := TRUE ;
		// add message data
		stFault.Active			:= TRUE 								;
		stFault.Discription		:= 'support not in safe (down) position';
		stFault.MessageNumber	:= E_MessageNumbers.FF_Collision 		;
		stFault.FaultType		:= E_FaultTypes.FF				;
		refFbFault.CmdAddFault( stFault );
	END_IF

// ====== Make sure support Moves down ======
	IF bActMovFwd 
	AND nActPos > nTriggerPosCheckDownFw 
	AND nActPos < nTriggerPosUpFw 
	AND NOT fbSensorClosed.bFcoInputActive THEN 
		// Set error to active (stop traverse axis) 
		bErrorActive := TRUE ;
		// add message data
		stFault.Active			:= TRUE 								;
		stFault.Discription		:= 'Emergency stop support cylinder not down';
		stFault.MessageNumber	:= E_MessageNumbers.FF_Collision 		;
		stFault.FaultType		:= E_FaultTypes.FF				;
		refFbFault.CmdAddFault( stFault );
	ELSIF bActMovRev 
	AND nActPos > nTriggerPosUprev
	AND nActPos < nTriggerPosCheckDownRe 
	AND NOT fbSensorClosed.bFcoInputActive THEN 
		// Set error to active (stop traverse axis) 
		bErrorActive := TRUE ;
		// add message data
		stFault.Active			:= TRUE 								;
		stFault.Discription		:= 'Emergency stop support cylinder not down';
		stFault.MessageNumber	:= E_MessageNumbers.FF_Collision 		;
		stFault.FaultType		:= E_FaultTypes.FF				;
		refFbFault.CmdAddFault( stFault );
 	END_IF
END_METHOD

METHOD Init_Support : BOOL
VAR_INPUT
	sInValveName		: STRING			:= 'valve'	; // Name of the cylinder ( used for fault handling and identification)
	nInValveNumber		: UDINT				:= 0		; // Cylinder identification number
	// Support data
	nInSupportPosition	: LREAL := 0 		; // possition of support cylinder in reference to the home position 
	nInSupportWidth		: LREAL := 100		; // width of support cylinder 
	// Traverse data 
	nInTravMaxAcc			: LREAL ; // traverse maximum acceleration 
	nInTravMaxDec			: LREAL ; // traverse maximum deceleration 
	nInTraverseLength		: LREAL	:= 550		; // Length of sewing head cart 
	nInTraverseFlagPosition	: LREAL	:= 0		; // position of flag in reference to edge of cart 
	// cart data
	nInHandCartLenght		: LREAL := 250		; // hand cart length [mm]
	nInHandCartClearance	: LREAL := 300		; // Clearance around cart in which support is down

	// safety values 	
	nInMinSafeDistanceDown: LREAL := 200		; // Minimum distance for support to move down
	// Command state
	eResetState		: E_ValveResetState := 0		; // Cylinder reset state variable (default is idle) 
	eSafeState		: E_ValveResetState	:= 0		; // Valve safe state
END_VAR
// ====== initi valve ======
	SUPER^.Init(nInValveNumber, eResetState, eSafeState);
	
// ====== Set support data =======
	nSupportPosition 	:= nInSupportPosition 	;
	nSupportWidth		:= nInSupportWidth 		;

// ====== Set traverse Data ======
	nTravMaxAcc				:= nInTravMaxAcc			;
	nTravMaxDec				:= nInTravMaxDec			;
	nTraverseLength 		:= nInTraverseLength		;
	nTraverseFlagPosition	:= nInTraverseFlagPosition 	;
	nMinSafeDistanceDown	:= nInMinSafeDistanceDown	;

// ===== set handcart data =====
	nHandCartLength 		:= nInHandCartLenght 		;
	nHandCartClearance		:= nInHandCartClearance		;

// ====== set feedback to true (support always has feedback) =======
	bIcfFbkClosedPresent 	:= TRUE ;
	bIcfFbkOpenPresent		:= TRUE ;
	
// ====== Check if init is done ======
END_METHOD

METHOD PUBLIC Mod_ManualControl : BOOL
VAR_INPUT
	eCmdCylinder : E_CylinderCmd ; // cylinder manual command	
END_VAR
bCmdManual := TRUE ;

CASE eCmdCylinder OF
	E_CylinderCmd.Cyl_Reset:
		CmdReset();
	E_CylinderCmd.Cyl_Hold:
		CmdHold();
	E_CylinderCmd.Cyl_Teach:
		CmdTeach();
	E_CylinderCmd.Cyl_Calculate:
		ExecCalc();
	E_CylinderCmd.Cyl_Expand:
		CmdOpen();
	E_CylinderCmd.Cyl_Retract:
		CmdClose();
	ELSE 
		RETURN;
END_CASE
END_METHOD

METHOD Mod_SupportDown : BOOL
VAR_INPUT
END_VAR
bCmdSupportDown := true ;
END_METHOD

END_FUNCTION_BLOCK

// Axis/FunctionBlocks/FB_Axis
FUNCTION_BLOCK FB_Axis EXTENDS FB_DevBase
VAR_IN_OUT
	//===== Axis Referance Udt =====
		AxisUdt : Udt_AxisData ; // Axis data udt
END_VAR
VAR	
	// ===== physical axis link =====
		AxisRef 	: Axis_Ref 		; // Referance to physical axis
		AxisState 	: ST_AxisStatus ; // Axis State indication directly from axis 
	// ===== Physical Homing signal =====
		IAxisHome AT %I* : BOOL ; // Axis homing sensor from PLC (if MC_DefaultHoming is used)
	// =============== Motion function blocks =================
		fbMcPower 		: MC_Power		;		// FB for enable and override
		fbMcReset 		: MC_Reset		;		// FB to reset axis
		fbSoeReset		: FB_SoEReset	; 		// FB to reset axis hardware
		fbMcHome		: MC_Home		;		// Fb to home Axis
		fbMcStop 		: MC_Stop		;		// FB to stop axis
		fbMcHalt		: MC_Halt		;		// FB to halt axis
		fbMcJog			: MC_Jog		;		// FB to Jog axis
		fbMCMoveRelative: MC_MoveRelative;		// FB to move relative
		fbMcMove		: MC_MoveAbsolute;		// FB to move axis (velocity movement)
		fbMcMoveVelo	: MC_MoveVelocity;		// FB to move with specified velocity until Next command is given
		fbMcMoveModulo	: MC_MoveModulo	;		// FB to move axis to modulo position
		fbGearInSlave	: MC_GearIn		;		// FB to gear axis to master 
		fbGearInDyn		: MC_GearInDyn	;		// Fb to gear axis dynamicly to master
		fbGearOutSlave	: MC_GearOut	;		// FB to decouple gearing
		
	// ============== Motion Status funtions ===================
		fbMcReadActualPosition 	: MC_ReadActualPosition ; // FB for reading actual position
		fbMcReadActualVelocity	: MC_ReadActualVelocity	; // FB for reading actual Velocity
		fbMcReadActualStatus	: MC_ReadStatus			; // Fb for reading actual status
		fbMcReadAxisError		: MC_ReadAxisError		; // FB for reading axis error 
		fbTimRemEnable			: TOF 					; // Timer for remove enable
		fbRtrigAxisError		: R_TRIG				; // FB for creating rising edge on Axis error
		fbRtrigDriveError		: R_TRIG				; // FB for creating rising edge on Drive error
		fbRtrigEnableError		: R_TRIG				; // FB for creating rising edge on drive error
	// ===== Message handling =====
		RTrigMessage : R_TRIG ;
		
END_VAR
VAR
	CmdVelocity	: UDT_AxVal	; // Command speed in degrees per second
	CmdAccel	: UDT_AxVal	; // Command acceleration
	CmdDecel	: UDT_AxVal	; // command deceleration
	PrevCommand		: E_AxisCmd ; // Previous axis Command
	NewCommand		: BOOL 		; // true when new command is given  

	EnableAxis		: BOOL 		; // Enable axis
	EnableAxisDelOff: BOOL 		; // Enable axis delayed off 
	EnableForward	: BOOL 		; // Enable forward motion
	EnableReverse	: BOOL 		; // Enable reverse movement
	EnableActive	: BOOL 		; // Enable active commands
	EnableError		: BOOL 		; // Enable error \
	EnableErrorId	: UDINT		; // Enable error id

	DriveFault		: BOOL 		; // Drive error 
	DriveFaultId	: UDINT 	; // Drive error Id

	AxisFault			: BOOL 		; // Axis Error Active
	AxisFaultId			: UDINT 	; // Axis Error Id
	AxisReady			: BOOL 		; // Axis is ready 

	RTrigAxisError	: BOOL 		; // Axis error rising edge
	RTrigDriveError	: BOOL 		; // Drive error rising edge
	RTrigEnableError: BOOL 		; // Enable error rising edge

	StepDone		: BOOL 		; // Axis step is done
	
	Act_SoeReset	: BOOL 		; // Hardware fault reset
	// ===== Function execute triggers =====
		Exec_Init 			: BOOL ; // Execute init 
		Exec_Reset			: BOOL ; // Execute reset
		Exec_Hold			: BOOL ; // Execute hold
		Exec_Home			: BOOL ; // Execute Home
		Exec_JogFwd			: BOOL ; // Execute Jog forward
		Exec_JogRev			: BOOL ; // Execute Jog reverse
		Exec_MoveRelative	: BOOL ; // Execute move relative
		Exec_MoveAbs		: BOOL ; // Execute move absolute reverse
		Exec_MoveModulo		: BOOL ; // Execute move modulo
		Exec_MoveVeloFwd	: BOOL ; // Execute move velocity forward
		Exec_MoveVeloRev	: BOOL ; // Execute move velocity reverse
		Exec_Hardstop		: BOOL ; // Execute hardstop
		Exec_Softstop		: BOOL ; // Execute Softstop
		Exec_GearAsSlave	: BOOL ; // Execute gear as slave
		Exec_GearSlaveDyn	: BOOL ; // Execute gear slave dynamic
		Exec_GearOutSlave	: BOOL ; // execute gear out slave
	// ===== Function ready feedback =====
		Fry_Init 			: BOOL ; // Execute init 
		Fry_Reset			: BOOL ; // Execute reset
		Fry_SoeReset		: BOOL ; // feedback ready reset hardware 
		Fry_Home			: BOOL ; // Execute Home
		Fry_Jog				: BOOL ; // Execute Jog forward
		Fry_MoveRelative	: BOOL ; // Execute move relative
		Fry_MoveAbs			: BOOL ; // Execute move absolute reverse
		Fry_MoveModulo		: BOOL ; // Execute move modulo
		Fry_MoveVeloFwd		: BOOL ; // Execute move velocity forward
		Fry_MoveVeloRev		: BOOL ; // Execute move velocity reverse
		Fry_GearAsSlave		: BOOL ; // Execute gear as slave
		Fry_GearSlaveDyn	: BOOL ; // Execute gear as dynamic slave
		Fry_GearOutSlave	: BOOL ; // Execute gear out slave
	// ===== Funtion errors =====
		Error_Init 			: BOOL ; // Error init 
		Error_Reset			: BOOL ; // Error reset
		Error_Hold			: BOOL ; // Error hold
		Error_Home			: BOOL ; // Error Home
		Error_JogFwd		: BOOL ; // Error Jog forward
		Error_JogRev		: BOOL ; // Error Jog reverse
		Error_MoveRelative	: BOOL ; // Error move relative
		Error_MoveAbs		: BOOL ; // Error move absolute reverse
		Error_MoveModulo	: BOOL ; // Error move modulo
		Error_MoveVeloFwd	: BOOL ; // Error move velocity forward
		Error_MoveVeloRev	: BOOL ; // Error move velocity reverse
		Error_Hardstop		: BOOL ; // Error hardstop
		Error_Softstop		: BOOL ; // Error Softstop
		Error_GearAsSlave	: BOOL ; // Error gear as slave
		Error_GearSlaveDyn	: BOOL ; // Error gear as dynamic slave
		Error_GearOutSlave	: BOOL ; // Error gear out slave
	// ===== Function Error Id's =====
		ErrorId_Init 		: UDINT ; // ErrorId init 
		ErrorId_Reset		: UDINT ; // ErrorId reset
		ErrorId_Hold		: UDINT ; // ErrorId hold
		ErrorId_Home		: UDINT ; // ErrorId Home
		ErrorId_JogFwd		: UDINT ; // ErrorId Jog forward
		ErrorId_JogRev		: UDINT ; // ErrorId Jog reverse
		ErrorId_MoveRelative: UDINT ; // ErrorId move relative
		ErrorId_MoveAbs		: UDINT ; // ErrorId move absolute forward
		ErrorId_MoveModulo	: UDINT ; // ErrorId move modulo
		ErrorId_MoveVeloFwd	: UDINT ; // ErrorId move velocity forward
		ErrorId_MoveVeloRev	: UDINT ; // ErrorId move velocity reverse
		ErrorId_Hardstop	: UDINT ; // ErrorId hardstop
		ErrorId_Softstop	: UDINT ; // ErrorId Softstop
		ErrorId_GearAsSlave	: UDINT ; // ErrorId gear as slave
		ErrorId_GearSlaveDyn: UDINT ; // ErrorId gear as dynamic slave
		ErrorId_GearOutSlave: UDINT ; // ErrorId gear out slave
END_VAR

// ===== Check safety =====
	// ***** when no safety active run command *****
		IF AxisUdt.AxisCmd = Ax_Reset OR bReset THEN 
			AxisUdt.AxisSafeCmd 	:= AxisUdt.AxisCmd			;
		ELSIF NOT AxisUdt.SafeCmdStop AND NOT AxisUdt.SafeCmdLimitVelo THEN 
			AxisUdt.AxisSafeCmd 	:= AxisUdt.AxisCmd			;
			AxisUdt.Velocity.SafeVal:= AxisUdt.Velocity.CmdVal 	;
			AxisUdt.Pos.SafeVal		:= AxisUdt.Pos.CmdVal 		;
		END_IF

	// ***** Axis emergency stop active *****
		IF AxisUdt.SafeCmdStop AND AxisUdt.AxisCmd <> Ax_Reset THEN 
			AxisUdt.AxisSafeCmd := Ax_HardStop ;
		END_IF
	
	// ***** Axis limit velocity *****		
		IF AxisUdt.SafeCmdLimitVelo AND ABS(AxisUdt.Velocity.ActVal) > AxisUdt.SafeVeloLimit + 50 THEN 
			AxisUdt.AxisSafeCmd 						:= Ax_SoftStop				;
			AxisUdt.Velocity.SafeVal					:= AxisUdt.SafeVeloLimit 	;
		ELSIF AxisUdt.SafeCmdLimitVelo THEN 
			AxisUdt.AxisSafeCmd 		:= AxisUdt.AxisCmd		;
			AxisUdt.Velocity.SafeVal	:= AxisUdt.SafeVeloLimit ;
			AxisUdt.Pos.SafeVal			:= AxisUdt.Pos.CmdVal 	;
			AxisUdt.SafeCmdLimitVelo 	:= FALSE 				;
		END_IF				
	
// ===== Check for new axis command =====
	IF 	AxisUdt.AxisSafeCmd <> PrevCommand THEN 
		NewCommand := TRUE ;
	ELSIF NOT AxisUdt.FcoGeared 
		AND (axisUdt.Pos.SafeVal <> AxisUdt.Pos.PrevVal 
		OR	AxisUdt.Velocity.SafeVal <> AxisUdt.Velocity.PrevVal) THEN 
		NewCommand := TRUE ;
	ELSE
		NewCommand := FALSE ;
	END_IF

	IF NewCommand AND NOT AxisUdt.ErrorActive THEN
		AxisUdt.Pos.PrevVal 		:= AxisUdt.Pos.SafeVal 		;
		AxisUdt.Velocity.PrevVal 	:= AxisUdt.Velocity.SafeVal 	;
		EnableActive 				:= FALSE 					; // disable active command
		StepDone					:= FALSE					; // step done set to false 	
	ELSIF AxisUdt.AxisSafeCmd = Ax_Reset AND AxisUdt.ErrorActive THEN 
		AxisUdt.AxisAct 			:= Ax_Reset 				;
		PrevCommand					:= AxisUdt.AxisSafeCmd			;
		StepDone 					:= FALSE 					;
		EnableActive				:= TRUE						; 		
	ELSIF NOT StepDone AND NOT AxisUdt.FcoGeared THEN 
		EnableActive 				:= TRUE 					; // Continue active command
	ELSIF Stepdone AND EnableActive THEN
		EnableActive				:= FALSE 					;
	ELSIF StepDone AND NOT EnableActive THEN
		AxisUdt.AxisAct 			:= Ax_Idle					;	// 
	END_IF

// ===== set Velocity command =====
	IF AxisUdt.IcfCommandSpeedRpm THEN
		CmdVelocity.AutoMax := Rpm_To_DegS(Rpm := AxisUdt.Velocity.AutoMax	);
		CmdVelocity.SafeVal	:= Rpm_To_DegS(Rpm := AxisUdt.Velocity.SafeVal	);
		CmdVelocity.HardMax	:= Rpm_To_DegS(Rpm := AxisUdt.Velocity.HardMax	);
		CmdVelocity.HomeMax	:= Rpm_To_DegS(Rpm := AxisUdt.Velocity.HomeMax	);
		CmdVelocity.ManMax	:= Rpm_To_DegS(Rpm := AxisUdt.Velocity.ManMax	);
		CmdVelocity.RefVal	:= Rpm_To_DegS(Rpm := AxisUdt.Velocity.RefVal	);
	ELSE
		CmdVelocity := AxisUdt.Velocity ;
	END_IF

// ===== Set acceleration and decelleration =====
	CmdAccel := axisudt.Accel ;
	CmdDecel := AxisUdt.Decel ;	
	
// ===== Enable both homing directions during motion =====
	IF AxisUdt.AxisAct = Ax_Home THEN ;
		Enablereverse 	:= TRUE ;
		EnableForward	:= TRUE	;
	ELSE
		EnableForward	:= AxisUdt.IcfEnableForward ;
		EnableReverse	:= AxisUdt.IcfEnableReverse	;
	END_IF

// ===== Remove enable when axis is idle for longer than 0.5 sec =====
	IF AxisUdt.CmdEnable AND (AxisUdt.AxisAct <> Ax_Idle OR AxisUdt.IcfAlwaysEnable) THEN
		EnableAxis := TRUE 	;
	ELSE
		EnableAxis := FALSE ;
	END_IF

	fbTimRemEnable (IN := EnableAxis, PT := AxisUdt.TimeDisableDelay, Q => EnableAxisDelOff);
	
	fbMcPower(	Axis			:= AxisRef , 
				Enable			:= EnableAxisDelOff, 
				Enable_Positive	:= EnableForward , 
				Enable_Negative	:= Enablereverse, 
				Override		:= 100, 
				BufferMode		:= Mc_Buffered, 
				Status			=> AxisUdt.FcoEnabled, 
				Busy			=> AxisUdt.ActBusy,  
				Error			=> EnableError, 
				ErrorID			=> AxisFaultId);

// ===== execute command =====
	CASE AxisUdt.AxisAct OF
		Ax_Idle:
			AxisUdt.ActBusy := FALSE ;
			AxisFault		:= FALSE ;
		Ax_Init:
			Exec_Init 	:= EnableActive ;
			AxisFault 	:= Error_Init 	;
			AxisFaultId	:= ErrorId_Init ;
			IF EnableActive AND Fry_Init THEN
				AxisUdt.FcoInit := TRUE ;
				StepDone := TRUE  ;
			END_IF
		Ax_Enable:
			AxisUdt.CmdEnable := TRUE	; // set enable command to true
			IF EnableActive THEN
				StepDone := AxisUdt.FcoEnabled ;
			END_IF
		Ax_Disable:
			AxisUdt.CmdEnable := FALSE	; // Set enable command to false
			IF EnableActive THEN
				StepDone := NOT AxisUdt.FcoEnabled ;
			END_IF 
		Ax_Reset: 
			Exec_Reset 	:= EnableActive ;
			AxisFault 	:= Error_Reset 	;
			AxisFaultId	:= ErrorId_Reset ;
			AxisUdt.CmdEnable 			:= FALSE ;
			AxisUdt.SafeCmdLimitVelo	:= FALSE ;
			IF NOT AxisRef.Status.Moving THEN 
				AxisUdt.SafeCmdStop := FALSE ;
			END_IF
			// ===== Reset all commands =====
				Exec_Init 			:= FALSE ; // Disable init 
				Exec_Hold			:= FALSE ; // Disable hold
				Exec_Home			:= FALSE ; // Disable Home
				Exec_JogFwd			:= FALSE ; // Disable Jog forward
				Exec_JogRev			:= FALSE ; // Disable Jog reverse
				Exec_MoveRelative	:= FALSE ; // Disable move relative
				Exec_MoveAbs		:= FALSE ; // Disable move absolute reverse
				Exec_MoveModulo		:= FALSE ; // Disable move modulo
				Exec_MoveVeloFwd	:= FALSE ; // Disable move velocity forward
				Exec_MoveVeloRev	:= FALSE ; // Disable move velocity reverse
				Exec_Hardstop		:= FALSE ; // Disable hardstop
				Exec_Softstop		:= FALSE ; // Disable Softstop
				Exec_GearAsSlave	:= FALSE ; // Disable gear as slave
				Exec_GearSlaveDyn	:= FALSE ; // Disable gear slave dynamic
				Exec_GearOutSlave	:= FALSE ; // Disable gear out slave
			IF AxisUdt.FcoReset AND EnableActive THEN
				StepDone := TRUE ;
			END_IF
		Ax_Hold:
			Exec_Hold 		:= EnableActive ;
			AxisFault 		:= Error_Hold 	;
			AxisFaultId		:= ErrorId_Hold ;
			IF EnableActive THEN
				StepDone 	:= NOT AxisUdt.ActBusy ;
			END_IF
		Ax_Home:
			IF AxisUdt.FcoEnabled THEN
				Exec_Home 	:= EnableActive ;
				AxisFault 	:= Error_Home 	;
				AxisFaultId	:= ErrorId_Home ;
			END_IF
			IF Fry_Home THEN
				AxisUdt.FcoHomed 	:= TRUE ;
				StepDone 			:= TRUE ;
			END_IF
		Ax_JogFwd:
			IF AxisUdt.FcoEnabled THEN
				Exec_JogFwd	:= EnableActive ;
				AxisFault 	:= Error_JogFwd	;
				AxisFaultId	:= ErrorId_JogFwd ;
			END_IF
		Ax_JogRev:
			IF AxisUdt.FcoEnabled THEN
				Exec_JogRev	:= EnableActive ;
				AxisFault 	:= Error_JogRev	;
				AxisFaultId	:= ErrorId_JogRev ;
			END_IF
		Ax_MoveRelative:
			IF AxisUdt.FcoEnabled THEN
				Exec_MoveRelative	:= EnableActive 		;
				AxisFault 			:= Error_MoveRelative	;
				AxisFaultId			:= ErrorId_MoveRelative ;
				AxisReady			:= Fry_MoveRelative 	;
				IF EnableActive THEN
					StepDone := Fry_MoveRelative ;
				END_IF
			END_IF
		Ax_MoveAbs:
			IF AxisUdt.FcoEnabled THEN
				Exec_MoveAbs	:= EnableActive 		;
				AxisFault 		:= Error_MoveAbs		;
				AxisFaultId		:= ErrorId_MoveAbs 	;
				AxisReady		:= Fry_MoveAbs	 		;
				IF EnableActive THEN
					StepDone := Fry_MoveAbs ;
				END_IF
			END_IF
		Ax_MoveModulo:
			IF AxisUdt.FcoEnabled THEN
				Exec_MoveModulo	:= EnableActive 		;
				AxisFault 		:= Error_MoveModulo		;
				AxisFaultId		:= ErrorId_MoveModulo 	;
				AxisReady		:= Fry_MoveModulo 		;
				IF EnableActive THEN
					StepDone := Fry_MoveModulo ;
				END_IF
			END_IF
		Ax_MoveVeloFwd:
			IF AxisUdt.FcoEnabled THEN
				Exec_MoveVeloFwd:= EnableActive 		;
				AxisFault 		:= Error_MoveVeloFwd	;
				AxisFaultId		:= ErrorId_MoveVeloFwd 	;
				AxisReady		:= Fry_MoveVeloFwd 		;
				IF EnableActive THEN
					StepDone := AxisUdt.ActAtVelo ;
				END_IF
			END_IF
		Ax_MoveVeloRev:
			IF AxisUdt.FcoEnabled THEN
				Exec_MoveVeloRev:= EnableActive 		;
				AxisFault 		:= Error_MoveVeloRev	;
				AxisFaultId		:= ErrorId_MoveVeloRev 	;
				AxisReady		:= Fry_MoveVeloRev 		;
				IF EnableActive THEN
					StepDone := AxisUdt.ActAtVelo ;
				END_IF
			END_IF	
		Ax_HardStop:
			Exec_Hardstop		:= EnableActive 	;
			CmdDecel.CmdVal		:= AxisUdt.Decel.HardMax ;
			AxisFault 			:= Error_Hardstop	;
			AxisFaultId			:= ErrorId_Hardstop	;
			IF EnableActive THEN
				StepDone 		:= AxisUdt.FcoStopped ;
			END_IF
		Ax_SoftStop:
			Exec_Softstop	:= EnableActive 	;
			AxisFault 		:= Error_Softstop	;
			AxisFaultId		:= ErrorId_Softstop	;
			IF EnableActive THEN
				StepDone := AxisUdt.FcoHeld 	;
			END_IF
		Ax_GearSlave:
			IF AxisUdt.FcoEnabled THEN
				Exec_GearAsSlave	:= EnableActive			;
				AxisFault 			:= Error_GearAsSlave	;
				AxisFaultId			:= ErrorId_GearAsSlave	;
			END_IF
				
			IF NOT EnableActive AND NOT Fry_GearAsSlave THEN 
				AxisUdt.AxisAct := Ax_GearOutSlave ;
			END_IF
		Ax_GearSlaveDyn:
			IF AxisUdt.FcoEnabled THEN
				Exec_GearSlaveDyn	:= EnableActive 		;
				AxisFault 			:= Error_GearSlaveDyn	;
				AxisFaultId			:= ErrorId_GearSlaveDyn	;
			END_IF 

			IF NOT  EnableActive AND Fry_GearSlaveDyn THEN 
				AxisUdt.AxisAct 	:= Ax_GearOutSlave ;
			END_IF
		Ax_GearOutSlave:
				Exec_GearAsSlave	:= FALSE 				;
				Exec_GearSlaveDyn	:= FALSE				;
				Exec_GearOutSlave 	:= TRUE 				;
 				AxisFault			:= Error_GearOutSlave	;
				AxisFaultId			:= ErrorId_GearOutSlave	;
			IF Fry_GearOutSlave THEN
				AxisUdt.FcoGeared 	:= FALSE 	;
				Exec_GearOutSlave 	:= FALSE	;
				StepDone			:= TRUE		;
			END_IF
		Ax_Maintenance:
			AxisUdt.CmdEnable 	:= TRUE  ; // Enable axis
			Exec_Init 			:= FALSE ; // Disable init 
			Exec_Reset			:= FALSE ; // Disable reset
			Exec_Hold			:= FALSE ; // Disable hold
			Exec_Home			:= FALSE ; // Disable Home
			Exec_JogFwd			:= FALSE ; // Disable Jog forward
			Exec_JogRev			:= FALSE ; // Disable Jog reverse
			Exec_MoveRelative	:= FALSE ; // Disable move relative
			Exec_MoveAbs		:= FALSE ; // Disable move absolute reverse
			Exec_MoveModulo		:= FALSE ; // Disable move modulo
			Exec_MoveVeloFwd	:= FALSE ; // Disable move velocity forward
			Exec_MoveVeloRev	:= FALSE ; // Disable move velocity reverse
			Exec_Hardstop		:= FALSE ; // Disable hardstop
			Exec_Softstop		:= FALSE ; // Disable Softstop
			Exec_GearAsSlave	:= FALSE ; // Disable gear as slave
			Exec_GearSlaveDyn	:= FALSE ; // Disable gear slave dynamic
			Exec_GearOutSlave	:= FALSE ; // Disable gear out slave
		ELSE // If an unknown axis command is given then go in error 
			AxisFault 	:= TRUE ;
			AxisFaultId	:= 100	;
	END_CASE
	
// ===== Check safety Stop =====
	IF NOT Exec_Hardstop AND AxisUdt.SafeCmdStop AND AxisUdt.AxisSafeCmd <> Ax_Reset THEN 
		Exec_Hardstop := AxisUdt.SafeCmdStop ; // Execute direct hardstop when safety commands it
		CmdDecel.CmdVal := AxisUdt.Decel.HardMax ;
	ELSIF Exec_Hardstop AND AxisRef.Status.HasBeenStopped AND NOT AxisUdt.SafeCmdStop THEN 
		Exec_Hardstop := FALSE ; 	
	END_IF

// ===== gear out when reset is active =====
	IF AxisUdt.AxisCmd = Ax_reset AND AxisRef.Status.Coupled THEN
		Exec_GearOutSlave := TRUE ;
	ELSIF NOT AxisRef.Status.Coupled THEN 
		Exec_GearOutSlave := FALSE ;
	END_IF 
	
// ===== Execute Motion functions =====
	Init(	Active 		:= Exec_Init, 
		 	Done		=> Fry_Init,
			Error 		=> Error_Init, 
		 	ErrorId		=> ErrorId_Init );
			
	Reset(	AxisRef		:= AxisRef,
			Active 		:= Exec_Reset, 
			Busy		=> AxisUdt.ActBusy,
			Moving		=> AxisUdt.ActMoving,
			Aborted		=> , 
			Done		=> AxisUdt.FcoReset, 
			Error 		=> Error_Reset, 
			ErrorId 	=> ErrorId_Reset );

	Hold(	AxisRef			:= AxisRef,
			CmdDeceleration	:= CmdDecel.CmdVal,
			Active 			:= Exec_Hold OR Exec_Softstop, 
			Busy			=> AxisUdt.ActBusy,
			Moving			=> AxisUdt.ActMoving,
			Aborted			=> , 
			Done			=> AxisUdt.FcoHeld, 
			Error 			=> Error_Hold, 
			ErrorId 		=> ErrorId_Hold );

	Home(	AxisRef			:= AxisRef,
			IHomeSwitch		:= IAxisHome,
			CmdHomingMode 	:= AxisUdt.CmdHomingMode,
			Posreferance	:= AxisUdt.Pos.RefVal, 
			Active 			:= Exec_Home, 
			Busy			=> AxisUdt.ActBusy,
			Moving			=> AxisUdt.ActMoving,
			Aborted			=> , 
			Done			=> Fry_Home, 
			Error 			=> Error_Home, 
			ErrorId 		=> ErrorId_Home);

	Jog(	AxisRef			:= AxisRef,
			CmdMode 		:= AxisUdt.CmdJogMode, 
			CmdPosition 	:= AxisUdt.Pos.SafeVal,
			CmdVelocity		:= CmdVelocity.SafeVal,
			CmdAcceleration	:= CmdAccel.CmdVal,
			CmdDeceleration	:= CmdDecel.CmdVal,
			ActiveFwd 		:= Exec_JogFwd,
			ActiveRev		:= Exec_JogRev, 
			Busy			=> AxisUdt.ActBusy,
			Moving			=> AxisUdt.ActMoving,
			Aborted			=> , 
			Done			=> Fry_Jog, 
			Error 			=> Error_JogFwd, 
			ErrorId 		=> ErrorId_JogFwd ); 

	MoveRelative(	AxisRef			:= AxisRef,
					CmdDistance		:= AxisUdt.Pos.SafeVal,
					CmdVelocity		:= CmdVelocity.SafeVal,
					CmdAcceleration	:= CmdAccel.CmdVal,
					CmdDeceleration	:= CmdDecel.CmdVal,
					Active			:= Exec_MoveRelative,
					BufferMode		:= AxisUdt.CmdBuffermode,
					Busy			=> AxisUdt.ActBusy,
					Moving			=> AxisUdt.ActMoving,
					Aborted			=> ,
					Done			=> Fry_MoveRelative,
					Error			=> Error_MoveRelative,
					ErrorId			=> ErrorId_MoveRelative );

	MoveAbs(	AxisRef			:= AxisRef,
				ActPosition		:= AxisUdt.Pos.ActVal,
				CmdPosition 	:= AxisUdt.Pos.SafeVal,
				CmdVelocity		:= CmdVelocity.SafeVal,
				CmdAcceleration := CmdAccel.CmdVal,
				CmdDeceleration	:= CmdDecel.CmdVal,
				Active 			:= Exec_MoveAbs, 
				BufferMode		:= AxisUdt.CmdBuffermode,
				Busy			=> AxisUdt.ActBusy,
				Moving			=> AxisUdt.ActMoving,
				Aborted			=> , 
				Done			=> Fry_MoveAbs, 
				Error 			=> Error_MoveAbs, 
				ErrorId 		=> ErrorId_MoveAbs ); 

	MoveModulo(	AxisRef			:= AxisRef,
				CmdPosition 	:= AxisUdt.Pos.SafeVal,
				CmdVelocity		:= CmdVelocity.SafeVal,
				CmdAcceleration := CmdAccel.CmdVal,
				CmdDeceleration	:= CmdDecel.CmdVal,
				Active 			:= Exec_MoveModulo, 
				BufferMode		:= AxisUdt.CmdBuffermode,
				Busy			=> AxisUdt.ActBusy,
				Moving			=> AxisUdt.ActMoving,
				Aborted			=> , 
				Done			=> Fry_MoveModulo, 
				Error 			=> Error_MoveModulo, 
				ErrorId 		=> ErrorId_MoveModulo );

	MoveVeloFwd(AxisRef			:= AxisRef,
				CmdVelocity		:= CmdVelocity.SafeVal,
				CmdAcceleration := CmdAccel.CmdVal,
				CmdDeceleration	:= CmdDecel.CmdVal,
				Active 			:= Exec_MoveVeloFwd, 
				BufferMode		:= AxisUdt.CmdBuffermode,
				AtVelocity		=> AxisUdt.ActAtVelo,
				Busy			=> AxisUdt.ActBusy,
				Moving			=> AxisUdt.ActMoving,
				Aborted			=> , 
				Done			=> Fry_MoveVeloFwd, 
				Error 			=> Error_MoveVeloFwd, 
				ErrorId 		=> ErrorId_MoveVeloFwd ); 

	MoveVeloRev(AxisRef			:= AxisRef,
				CmdVelocity		:= CmdVelocity.SafeVal,
				CmdAcceleration := CmdAccel.CmdVal,
				CmdDeceleration	:= CmdDecel.CmdVal,
				Active 			:= Exec_MoveVeloRev, 
				BufferMode		:= AxisUdt.CmdBuffermode,
				AtVelocity		=> AxisUdt.ActAtVelo,
				Busy			=> AxisUdt.ActBusy,
				Moving			=> AxisUdt.ActMoving,
				Aborted			=> , 
				Done			=> Fry_MoveVeloRev, 
				Error 			=> Error_MoveVeloRev, 
				ErrorId 		=> ErrorID_MoveVeloRev );

	Stop(	AxisRef		:= AxisRef,
			CmdDecel 	:= CmdDecel.CmdVal,
			Active 		:= Exec_Hardstop, 
			Busy		=> AxisUdt.ActBusy,
			Moving		=> AxisUdt.ActMoving,
			Aborted		=> , 
			Done		=> axisUdt.FcoStopped, 
			Error 		=> Error_Hardstop, 
			ErrorId 	=> ErrorId_Hardstop );

	GearAsSlave ( 	SlaveAxisRef	:= AxisRef,	
					MasterAxisRef 	:= AxisUdt.MasterAxisRef,
					Numerator		:= AxisUdt.GearSlaveRev,		
					Denominator		:= AxisUdt.GearMasterRev, 
					Active		  	:= Exec_GearAsSlave,  
					InGear			=> Fry_GearAsSlave,
					Busy			=> AxisUdt.ActBusy,
					Moving			=> AxisUdt.ActMoving,
					Aborted			=> , 
					Error 			=> Error_GearAsSlave,
					ErrorId			=> ErrorId_GearAsSlave );

	GearSlaveDyn(	SlaveAxisRef	:= AxisRef,	
					MasterAxisRef 	:= AxisUdt.MasterAxisRef,
					Numerator		:= AxisUdt.GearSlaveRev,		
					Denominator		:= AxisUdt.GearMasterRev,
					ReverseSlave	:= AxisUdt.ReverseSlave, 
					Active		  	:= Exec_GearSlaveDyn,  
					InGear			=> Fry_GearSlaveDyn,
					Busy			=> AxisUdt.ActBusy,
					Moving			=> AxisUdt.ActMoving,
					Aborted			=> , 
					Error 			=> Error_GearSlaveDyn,
					ErrorId			=> ErrorId_GearSlaveDyn );

	GearOutSlave(	SlaveAxisRef	:= AxisRef,
					Active			:= Exec_GearOutSlave,
					Busy			=> AxisUdt.ActBusy,
					Done			=> Fry_GearOutSlave,
					Error			=> Error_GearOutSlave,
					ErrorId			=> ErrorId_GearOutSlave );
					
// ===== get Actual axis values =====
	GetActVal(	AxisUdt := AxisUdt,
				Error 	=> DriveFault,
				ErrorId	=> DriveFaultId);
// ===== Get actual axis Status =====
		AxisUdt.FcoGeared := AxisRef.Status.Coupled ;

// ===== Fault and message handling =====	
	// ***** Create error string *****
		fbRtrigAxisError	(CLK := AxisFault	, Q => RTrigAxisError	);
		fbRtrigDriveError	(CLK := DriveFault	, Q => RTrigDriveError	);
		fbRtrigEnableError	(CLK := EnableError	, Q => RTrigEnableError );
	
		IF RTrigAxisError THEN 
			stFault.Discription	:= Concat(', Axis Fault: ', UDINT_TO_STRING(AxisFaultId)) ;
		ELSIF RTrigDriveError THEN 
			stFault.Discription 	:= Concat(', Drive Fault: ', UDINT_TO_STRING(DriveFaultId));
		ELSIF RTrigEnableError THEN
			stFault.Discription	:= Concat(', EnableFault: ', UDINT_TO_STRING(EnableErrorId)) ;
		END_IF
		
	// ***** Set Axis error *****
		IF AxisFault THEN
			AxisUdt.errorActive 	:= TRUE ;
			stFault.MessageNumber 	:= E_MessageNumbers.FF_AxisFault ;
			stFault.Discription 	:= Concat(', Axis Fault: ', UDINT_TO_STRING(AxisFaultId));
			stFault.FaultType 		:= E_FaultTypes.FF ;
		ELSIF DriveFault THEN
			AxisUdt.errorActive 	:= TRUE ;
			stFault.MessageNumber 	:= E_MessageNumbers.FF_DriveFault ;
			stFault.Discription 	:= Concat(', Drive Fault: ', UDINT_TO_STRING(DriveFaultId)) ;
			stFault.FaultType 		:= E_FaultTypes.FF ;
		ELSIF EnableError THEN
			AxisUdt.errorActive 	:= TRUE ;
			stFault.MessageNumber 	:= E_MessageNumbers.CF_FeedbackFault ;
			stFault.Discription 	:= Concat(', EnableFault: ', UDINT_TO_STRING(EnableErrorId)) ;
			stFault.FaultType 		:= E_FaultTypes.CF ;
		ELSIF AxisUdt.AxisSafeCmd = Ax_Reset THEN
			AxisFault			:= FALSE ; 
			AxisUdt.ErrorActive := FALSE ;
		ELSE
			AxisUdt.ErrorActive := FALSE ;
		END_IF
		
	// ***** write message data to higher level *****
	
	IF AxisUdt.ErrorActive THEN 
		stFault.Active 			:= TRUE ;
		stFault.ComponentType 	:= E_ComponentTypes.Axis ;
		stFault.LocationName	:= 'Powerline main axis ' ;
		stFault.LocationNumber	:= INT_TO_UDINT( AxisUdt.AxisNumber)	;
		refFbFault.CmdAddFault( stFault );
	END_IF

// ===== Set Axis ready bit =====
	AxisUdt.FcoReady	:= StepDone	;

	IF AxisUdt.AxisAct = Ax_Idle THEN 
		AxisUdt.FcoIdle	:= TRUE 	;
	ELSE
		AxisUdt.FcoIdle	:= FALSE 	;
	END_IF

// ===== Set Command to active =====
		IF NOT AxisUdt.ErrorActive AND NOT AxisUdt.FcoGeared AND AxisUdt.AxisSafeCmd <> Ax_Reset THEN
			PrevCommand		:= AxisUdt.AxisSafeCmd ;
			AxisUdt.AxisAct := AxisUdt.AxisSafeCmd ;
		ELSIF AxisUdt.AxisCmd = Ax_reset THEN 
			IF AxisRef.Status.Moving THEN 
				AxisUdt.SafeCmdStop := TRUE ;
			END_IF
			PrevCommand		:= Ax_reset ;
			AxisUdt.AxisAct := AxisUdt.AxisSafeCmd ;
		END_IF

// ==== Set command active bit when act = cmd =====
	IF AxisUdt.AxisAct = AxisUdt.AxisCmd
	AND AxisUdt.Velocity.SafeVal = AxisUdt.Velocity.CmdVal
	AND AxisUdt.Pos.SafeVal		= AxisUdt.Pos.CmdVal THEN 
		AxisUdt.FcoCmdActive	:= TRUE ;
	ELSE
		AxisUdt.FcoCmdActive	:= FALSE ;
	END_IF

(* gear axis as slave *)
METHOD PRIVATE GearAsSlave : BOOL
VAR_IN_OUT
	SlaveAxisRef	: Axis_Ref	; // Slave axis referance
	MasterAxisRef 	: Axis_Ref 	; // Master axis referance 
END_VAR
VAR_INPUT
	Numerator		: LREAL		; // gear ratio numeration (slave axis rev)
	Denominator		: UINT		; // Gear ratio denominator (master axis rev) 
	Active		  	: BOOL 		; // Activate gearing  
END_VAR
VAR_OUTPUT
	InGear			: BOOL 		; // axis is geared
	Busy			: BOOL 		; // axis is busy
	Moving			: BOOL 		; // axis is moving
	Aborted			: BOOL 		; // Axis command was aborted
	Error 			: BOOL 		; // Function error active
	ErrorId			: UDINT 	; // Error Id number
END_VAR
// ===== Gear axis in =====
	fbGearInSlave(	Master:= MasterAxisRef , 
					Slave:= SlaveAxisRef, 
					Execute:= Active , 
					RatioNumerator:= Numerator, 
					RatioDenominator:= Denominator, 
					InGear=> InGear, 
					Busy=> Busy, 
					Active=> Moving, 
					CommandAborted=> Aborted, 
					Error=>	Error , 
					ErrorID=> ErrorId );
END_METHOD

(* gear axis as slave *)
METHOD PRIVATE GearOutSlave : BOOL
VAR_IN_OUT
	SlaveAxisRef	: Axis_Ref	; // Slave axis referance
END_VAR
VAR_INPUT
	Active		  	: BOOL 		; // Activate gearing  
END_VAR
VAR_OUTPUT
	Busy			: BOOL 		; // axis is busy
	Aborted			: BOOL 		; // Axis command was aborted
	Done			: BOOL 		; // Axis command was executed succesfully 
	Error 			: BOOL 		; // Function error active
	ErrorId			: UDINT 	; // Error Id number
END_VAR
// ===== Gear axis out =====
fbGearOutSlave(	Slave := SlaveAxisRef,
				Execute := Active,
				Options	:=,
				Done	=> Done,
				Busy	=> Busy,
				Error	=> Error,
				ErrorID	=> ErrorId
				);
END_METHOD

METHOD PRIVATE GearSlaveDyn : BOOL
VAR_IN_OUT
	SlaveAxisRef	: Axis_Ref	; // Slave axis referance
	MasterAxisRef 	: Axis_Ref 	; // Master axis referance 
END_VAR
VAR_INPUT
	Numerator		: LREAL		; // gear ratio numeration (slave axis rev)
	Denominator		: UINT		; // Gear ratio denominator (master axis rev) 
	ReverseSlave	: BOOL 		; // Reverse slave axis relative to master
	Active		  	: BOOL 		; // Activate gearing  
END_VAR
VAR_OUTPUT
	InGear			: BOOL 		; // axis is geared
	Busy			: BOOL 		; // axis is busy
	Moving			: BOOL 		; // axis is moving
	Aborted			: BOOL 		; // Axis command was aborted
	Error 			: BOOL 		; // Function error active
	ErrorId			: UDINT 	; // Error Id number
END_VAR
VAR
	Gearfactor : LREAL ;
END_VAR
// ===== Calculate gear factor =====
	IF Active AND Denominator <> 0 THEN
		Gearfactor := Numerator / UDINT_TO_LREAL(Denominator);
	END_IF

	IF ReverseSlave THEN
		Gearfactor := Gearfactor * -1;
	END_IF


// ==== Gear in Dynamically ====
	fbGearInDyn(	Master			:= MasterAxisRef , 
					Slave			:= SlaveAxisRef, 
					Enable			:= Active,
					GearRatio 		:= Gearfactor,
					Acceleration	:= 0,
					Deceleration	:= 0,
					Jerk			:= 0,
					BufferMode		:=,
					Options			:=,
					InGear			=> InGear, 
					Busy			=> Busy, 
					Active			=> Moving, 
					CommandAborted	=> Aborted, 
					Error			=>	Error , 
					ErrorID			=> ErrorId );
END_METHOD

(* Get Actual axis values *)
METHOD PRIVATE GetActVal : BOOL
VAR_IN_OUT
	//===== Axis Referance Udt =====
		AxisUdt : Udt_AxisData ; // Axis data udt
END_VAR
VAR_OUTPUT
	Valid 	: BOOL ; // read is valid
	Error 	: BOOL ; // Axis Error active
	ErrorID	: Udint ; // Axis error ID
END_VAR
VAR 
	ErrorInternal	: BOOL ; // error
	actPos		 	: LREAL ; // temporary axis pos
	actVel			: LREAL ; // Temporary Velocity
	ErrorIdInternal	: UDINT ; // Error Id number
END_VAR
// ===== Read error status =====
	fbMcReadAxisError(Axis := AxisRef,Enable := TRUE, Valid => Valid, Error => ErrorInternal, ErrorId => errorIdInternal);
	IF Valid THEN
		Error 	:= ErrorInternal ;
		ErrorID	:= ErrorIdInternal;
	END_IF

// ===== Read actual position =====
	fbMcReadActualPosition(Axis := AxisRef, Enable := TRUE, Valid => Valid,Position => ActPos) ;
	IF Valid THEN
		AxisUdt.Pos.ActVal := ActPos ;
		AxisUdt.Pos.ActModulo := AxisRef.NcToPlc.ModuloActPos	;	
	END_IF

// ===== Get axis state information =====
	fbMcReadActualStatus (Axis := AxisRef, Enable := TRUE, Status => AxisState);
		
// ===== Read actual velocity =====
	fbMcreadactualVelocity(Axis := AxisRef, Enable := TRUE, Valid => Valid,ActualVelocity => ActVel);
	IF valid AND AxisUdt.IcfCommandSpeedRpm THEN
		AxisUdt.Velocity.ActVal := DegS_To_Rpm(DegS := ActVel);
	ELSE 
		AxisUdt.Velocity.ActVal := actVel ;
	END_IF
	
// ===== Get Actual values from physical axis =====
	AxisUdt.Accel.ActVal		:= AxisRef.NcToPlc.ActAcc	; // Get Actual acceleration
	AxisUdt.Torque.ActVal		:= AxisRef.NcToPlc.ActTorque; // Get Actual torque
END_METHOD

(* bring axis to controlled stop and hold it until next command *)
METHOD private Hold : BOOL
VAR_IN_OUT
	AxisRef	: Axis_Ref ; // Axis referance
END_VAR
VAR_INPUT
	CmdDeceleration : LREAL ; // command deceleration 
	Active	: BOOL ; // activate movement 
END_VAR
VAR_OUTPUT
	Busy	: BOOL	; // axis is busy
	Moving	: BOOL	; // axis is moving
	Aborted	: BOOL	; // Axis command was aborted
	Done	: BOOL	; // Axis command was executed succesfully 
	Error 	: BOOL 	; // Function error active
	ErrorId	: UDINT ; // Error Id number
END_VAR
//===== Halt Axis =====
	fbMcHalt(	Axis		:= AxisRef , 
				Execute		:= Active, 
				Deceleration:= CmdDeceleration , 
				Jerk		:= , 
				BufferMode	:= MC_Aborting,  
				Done		=> Done , 
				Busy		=> Busy , 
				CommandAborted=> Aborted , 
				Error		=> Error, 
				ErrorID		=> ErrorId
				);
END_METHOD

(* Home Axis and set position to referance value *)
METHOD PRIVATE  Home : BOOL
VAR_IN_OUT
	AxisRef			: Axis_Ref 		; // Axis referance 
END_VAR
VAR_INPUT
	IHomeSwitch		: BOOL 			; // homing position input 
	CmdHomingMode 	: MC_HomingMode ; // Axis Homing Mode
	PosReferance  	: LREAL 		; // Home position is set to referance value Default is 0 
	Active			: BOOL 			; // activate movement 
END_VAR
VAR_OUTPUT
	Busy	: BOOL	; // axis is busy
	Moving	: BOOL	; // axis is moving
	Aborted	: BOOL	; // Axis command was aborted
	Done	: BOOL	; // Axis command was executed succesfully 
	Error 	: BOOL 	; // Function error active
	ErrorId	: UDINT ; // Error Id number
END_VAR
// ===== home Axis =====
fbMcHome(	Axis			:= AxisRef , 
			Execute			:= Active , 
			Position		:= , 
			HomingMode		:= CmdHomingMode ,
			bCalibrationCam := IHomeSwitch, 
			Done			=> Done , 
			Busy			=> Busy, 
			CommandAborted	=> Aborted , 
			Error			=> Error , 
			ErrorID			=> ErrorId );
END_METHOD

(* Axis initialisation *)
METHOD PRIVATE  Init : BOOL
VAR_INPUT
	Active	: BOOL ; // activate movement 
END_VAR
VAR_OUTPUT
	Done	: BOOL 	; // Axis command was executed succesfully
	Error 	: BOOL 	; // Function error active
	ErrorId	: UDINT ; // Error Id number
END_VAR
IF Active THEN 
	// ===== set init to done =====
		Done := TRUE ;
END_IF
END_METHOD

(* Jog axis forward *)
METHOD PRIVATE Jog : BOOL
VAR_IN_OUT
		AxisRef	: Axis_Ref ; // Axis referance 
END_VAR
VAR_INPUT
	ActiveFwd	: BOOL 		; // Activate movement jog forward
	ActiveRev	: BOOL 		; // Activate movement Jog reverse
	CmdMode		: E_Jogmode ; // Jog mode [slow, fast, continuous, inching, modulo]
	CmdPosition	: LREAL		; // position increment distance when in inching, stop position when in modulo
	CmdVelocity : LREAL		; // Jog velocity [0 = standard velocity]
	CmdAcceleration	: LREAL	; // Jog Acceleration
	CmdDeceleration	: LREAL	; // Jog deceleration
END_VAR
VAR_OUTPUT
	Busy	: BOOL	; // axis is busy
	Moving	: BOOL	; // axis is moving
	Aborted	: BOOL	; // Axis command was aborted
	Done	: BOOL	; // Axis command was executed succesfully 
	Error 	: BOOL 	; // Function error active
	ErrorId	: UDINT ; // Error Id number
END_VAR

// ===== Jog Axis =====
fbMcJog(	Axis			:= AxisRef, 
			JogForward		:= ActiveFwd, 
			JogBackwards	:= ActiveRev, 
			Mode			:= CmdMode, 
			Position		:= CmdPosition , 
			Velocity		:= CmdVelocity, 
			Acceleration	:= CmdAcceleration, 
			Deceleration	:= CmdDeceleration, 
			Jerk			:= 0, 
			Done			=> Done, 
			Busy			=> Busy, 
			Active			=> Moving, 
			CommandAborted	=> Aborted , 
			Error			=> Error , 
			ErrorID			=> ErrorId );
END_METHOD

(* Move axis reverse for set distance *)
METHOD PRIVATE MoveAbs : BOOL
VAR_IN_OUT
	AxisRef	: Axis_Ref ; // Axis referance 
END_VAR
VAR_INPUT
	ActPosition		: LREAL; // Actual axis position
	CmdPosition 	: LREAL; // Command position
	CmdVelocity 	: LREAL; // Move velocity
	CmdAcceleration	: LREAL; // Move Acceleration
	CmdDeceleration	: LREAL; // Move deceleration
	Active			: BOOL ; // activate movement 
	BufferMode		: MC_BufferMode ; // Buffermode used for command transition  
	
END_VAR
VAR_OUTPUT
	Busy	: BOOL	; // axis is busy
	Moving	: BOOL	; // axis is moving
	Aborted	: BOOL	; // Axis command was aborted
	Done	: BOOL	; // Axis command was executed succesfully 
	Error 	: BOOL 	; // Function error active
	ErrorId	: UDINT ; // Error Id number
END_VAR
// ===== Move instruction =====
	fbMcMove(	Axis:= AxisRef , 
				Execute:= Active, 
				Position:= CmdPosition, 
				Velocity:= CmdVelocity, 
				Acceleration:= CmdAcceleration, 
				Deceleration:= CmdDeceleration, 
				Jerk:= 0, 
				BufferMode:= BufferMode , 
				Options:= , 
				Done=> Done, 
				Busy=> Busy, 
				Active=> Moving, 
				CommandAborted=> Aborted , 
				Error=> Error, 
				ErrorID=> ErrorId );
END_METHOD

(* Move axis to set position on 360deg scale (used for needle positioning) *)
METHOD PRIVATE MoveModulo : BOOL
VAR_IN_OUT
	AxisRef	: Axis_Ref ; // Axis referance 
END_VAR
VAR_INPUT
	CmdPosition 	: LREAL; // Command position
	CmdVelocity 	: LREAL; // Move velocity
	CmdAcceleration	: LREAL; // Move Acceleration
	CmdDeceleration	: LREAL; // Move deceleration
	Active			: BOOL ; // activate movement 
	BufferMode		: MC_BufferMode ; // Buffermode used for command transition  

END_VAR
VAR_OUTPUT
	Busy	: BOOL	; // axis is busy
	Moving	: BOOL	; // axis is moving
	Aborted	: BOOL	; // Axis command was aborted
	Done	: BOOL	; // Axis command was executed succesfully 
	Error 	: BOOL 	; // Function error active
	ErrorId	: UDINT ; // Error Id number
END_VAR
// ===== move modulo =====
fbMcMoveModulo(	Axis:= AxisRef , 
				Execute:= Active, 
				Position:= CmdPosition, 
				Velocity:= CmdVelocity, 
				Acceleration:= CmdAcceleration, 
				Deceleration:= CmdDeceleration, 
				Jerk:= 0, 
				Direction:= mc_Positive_Direction, 
				BufferMode:= BufferMode, 
				Options:= , 
				Done=> Done , 
				Busy=> Busy, 
				Active=> Moving, 
				CommandAborted=> Aborted, 
				Error=> Error, 
				ErrorID=> ErrorId);
END_METHOD

(* Move axis relative to current position *)
METHOD PRIVATE MoveRelative : BOOL
VAR_IN_OUT
	AxisRef	: Axis_Ref ; // Axis referance 
END_VAR
VAR_INPUT
	CmdDistance 	: LREAL; // Command position
	CmdVelocity 	: LREAL; // Move velocity
	CmdAcceleration	: LREAL; // Move Acceleration
	CmdDeceleration	: LREAL; // Move deceleration
	Active			: BOOL ; // activate movement
	BufferMode		: MC_BufferMode ; // Buffermode used for command transition  
 
END_VAR
VAR_OUTPUT
	Busy	: BOOL	; // axis is busy
	Moving	: BOOL	; // axis is moving
	Aborted	: BOOL	; // Axis command was aborted
	Done	: BOOL	; // Axis command was executed succesfully 
	Error 	: BOOL 	; // Function error active
	ErrorId	: UDINT ; // Error Id number
END_VAR
fbMCMoveRelative(	Axis			:= AxisRef ,
					Execute			:= Active ,
					Distance		:= CmdDistance ,
					Velocity		:= CmdVelocity,
					Acceleration	:= CmdAcceleration,
					Deceleration	:= CmdDeceleration,
					Jerk			:= 0,
					BufferMode		:= BufferMode,
					Options			:= ,
					Done			=> Done,
					Busy			=> Busy,
					Active			=> Moving,
					CommandAborted	=> Aborted,
					Error			=> Error,
					ErrorID			=> ErrorId
				);
END_METHOD

(* Move with set velocity until commanded otherwise *)
METHOD PRIVATE MoveVeloFwd : BOOL
VAR_IN_OUT
	AxisRef	: Axis_Ref ; // Axis referance 
END_VAR
VAR_INPUT
	CmdVelocity 	: LREAL; // Move velocity
	CmdAcceleration	: LREAL; // Move Acceleration
	CmdDeceleration	: LREAL; // Move deceleration
	Active			: BOOL ; // activate movement
	BufferMode		: MC_BufferMode ; // Buffermode used for command transition  
	
END_VAR
VAR_OUTPUT
	AtVelocity : BOOL ; // Axis is at velocity
	Busy	: BOOL	; // axis is busy
	Moving	: BOOL	; // axis is moving
	Aborted	: BOOL	; // Axis command was aborted
	Done	: BOOL	; // Axis command was executed succesfully 
	Error 	: BOOL 	; // Function error active
	ErrorId	: UDINT ; // Error Id number
END_VAR
// ===== move with set velocity =====
fbMcMoveVelo(	Axis:= AxisRef, 
				Execute:= Active, 
				Velocity:= CmdVelocity, 
				Acceleration:= CmdAcceleration, 
				Deceleration:= CmdDeceleration, 
				Jerk:= 0, 
				Direction:= MC_Positive_direction, 
				BufferMode:= BufferMode , 
				Options:= , 
				InVelocity=> AtVelocity, 
				Busy=> Busy, 
				Active=> Moving, 
				CommandAborted=> Aborted , 
				Error=> Error, 
				ErrorID=> Errorid );
END_METHOD

(* Move with set velocity routine *)
METHOD PRIVATE MoveVeloRev : BOOL
VAR_IN_OUT
	AxisRef	: Axis_Ref ; // Axis referance 
END_VAR
VAR_INPUT
	CmdVelocity 	: LREAL; // Move velocity
	CmdAcceleration	: LREAL; // Move Acceleration
	CmdDeceleration	: LREAL; // Move deceleration
	Active			: BOOL ; // activate movement
	BufferMode		: MC_BufferMode ; // Buffermode used for command transition 
END_VAR
VAR_OUTPUT
	AtVelocity : BOOL ; // Axis is at velocity
	Busy	: BOOL	; // axis is busy
	Moving	: BOOL	; // axis is moving
	Aborted	: BOOL	; // Axis command was aborted
	Done	: BOOL	; // Axis command was executed succesfully 
	Error 	: BOOL 	; // Function error active
	ErrorId	: UDINT ; // Error Id number
END_VAR
// ===== move with set velocity =====
fbMcMoveVelo(	Axis:= AxisRef, 
				Execute:= Active, 
				Velocity:= CmdVelocity, 
				Acceleration:= CmdAcceleration, 
				Deceleration:= CmdDeceleration, 
				Jerk:= 0, 
				Direction:= MC_Negative_direction, 
				BufferMode:= BufferMode , 
				Options:= , 
				InVelocity=> AtVelocity, 
				Busy=> Busy, 
				Active=> Moving, 
				CommandAborted=> Aborted , 
				Error=> Error, 
				ErrorID=> Errorid );
END_METHOD

(* reset axis faults *)
METHOD PRIVATE Reset : BOOL
VAR_IN_OUT
	AxisRef	: Axis_Ref ; // Axis referance 
END_VAR
VAR_INPUT
	Active	: BOOL ; // activate movement 
END_VAR
VAR_OUTPUT
	SoeBusy	: BOOL  ; // Axis hardware reset busy
	Busy	: BOOL	; // axis is busy
	Moving	: BOOL	; // axis is moving
	Aborted	: BOOL	; // Axis command was aborted
	Done	: BOOL	; // Axis command was executed succesfully 
	Error 	: BOOL 	; // Function error active
	ErrorId	: UDINT ; // Error Id number
END_VAR
// ===== Reset axis hardware =====
fbSoeReset(	NetId 	:=,
			Execute := Active,
			Axis	:= AxisRef,
			Timeout := T#10S,
			Busy	=> SoeBusy,
			Error	=> Error,
			AdsErrId=> ErrorId );

IF NOT fbSoeReset.Busy THEN 
// ===== Reset Axis =====
fbMcReset(	Axis:= AxisRef , 
			Execute:= Active, 
			Done=> Done, 
			Busy=> Busy, 
			Error=> Error, 
			ErrorID=> ErrorId );
END_IF

IF NOT fbSoeReset.Busy AND fbMcReset.Done THEN 
	Done := TRUE ;
ELSE
	Done := FALSE ;
END_IF
END_METHOD

(* Stop axis routine *)
METHOD PRIVATE Stop : BOOL
VAR_IN_OUT
	AxisRef	: Axis_Ref ; // Axis referance 
END_VAR
VAR_INPUT
	CmdDecel: LREAL	; // commanded deceleration value
	Active	: BOOL 	; // activate movement 
END_VAR
VAR_OUTPUT
	Busy	: BOOL 	; // axis is busy
	Moving	: BOOL 	; // axis is moving
	Aborted	: BOOL 	; // Axis command was aborted
	Done	: BOOL 	; // Axis command was executed succesfully 
	Error 	: BOOL 	; // Function error active
	ErrorId	: UDINT ; // Error Id number
END_VAR
fbMcStop(	Axis:= AxisRef, 
			Execute:= Active, 
			Deceleration:= CmdDecel, 
			Jerk:= 0, 
			Done=> Done, 
			Busy=> Busy, 
			CommandAborted=> , 
			Error=> Error, 
			ErrorID=> ErrorId
		);
END_METHOD

END_FUNCTION_BLOCK

// Axis/FunctionBlocks/Fb_AxisNew
FUNCTION_BLOCK PUBLIC Fb_AxisNew EXTENDS FB_DevBase
VAR_INPUT
	// ===== General Function input =====
		fCmdAcc			: LREAL := 15000;
		fCmdDecc		: LREAL := 15000; 
	// ===== Master Axis =====
		refMasterAxis	: REFERENCE TO AXIS_REF ; // Master axis reference (if applicable)
		bReverseSlave	: BOOL 	:= FALSE; // Reverse slave axis relative to master
		fCmdGearRatio	: LREAL := 1 ; // Gear ratio Master/Slave (1/Ratio) 
END_VAR
VAR_OUTPUT
	// ====== State indications =======
		bInitDone		: BOOL 	:= FALSE;
		bHomed			: BOOL 	:= FALSE; 
		bError 			: BOOL 	:= FALSE;
		bStopped		: BOOL 	:= FALSE;
		bGearedAsSlave	: BOOL 	:= FALSE;
		bVelocityLimited: BOOL 	:= FALSE;  
		bIdle			: BOOL 	:= FALSE;
		bErrorId		: BOOL 	:= FALSE;
		fVelocity		: LREAL	:= 0	; // Axis velocity [rpm on units/sec] depending on config
	// ====== axis reference ======
		AxisRef			: AXIS_REF	; // Axis reference to hardware 
	// ====== Axis Settings ======
		fMaxVelo		: LREAL := 0 ; // Axis Maximum velocity
		fMaxAcc			: LREAL := 0 ; // Axis Maximum cceleration
		fMaxDec			: LREAL := 0 ; // axis Maxium deceleration 
	
		fSafeVeloLimit	: LREAL	:= 200; // Safe velocity limit 
		tDisableDelay	: TIME 	:= T#500MS ;
	// ==== Axis data ====
		fEncoderTurnoverValue	: LREAL ;   
END_VAR
VAR // Axis configuration 
	// ===== HW Config Bits =====
		bIcfCmdVelocityRpm	: BOOL ; // input speeds in Rpm
		bIcfEnableForward 	: BOOL ; // Enable forward motion
 		bIcfEnablereverse	: BOOL ; // Enable reverse motion
		bIcfAlwaysEnable	: BOOL ; // 1 = Axis always enabled, 0 = Axis disabled at Idle 
		bIcfSimulationMode	: BOOL := FALSE ; // Simulation mode is active [default set to False] 
	// ===== Internal motion values ======
		fHomePosition		: LREAL := 0 ; // set position at homing
	// Command Modes
		mcHomingMode 		: MC_HomingMode := MC_direct ; // Homing Mode ( MC_DefaultHoming, MC_Direct, MC_ForceCallibration, MC_ResetCallibration)
	// Values from system
		McReadSysVelo		: MC_ReadParameter		; // Read Acceleration parameter from drive 
		McReadSysAcc		: MC_ReadParameter		; // Read Acceleration parameter from drive 
		McReadSysDec		: MC_ReadParameter		; // Read Acceleration parameter from drive 
END_VAR
VAR	// ====== Axis enable =====
		bCmdEnableAxis 		: BOOL := FALSE ; // Command to enable the axis (External)
		bInternalEnable		: BOOL := FALSE ; // internal enable command (turns off after set time, and on at new motion command
		TofIntAxisEnable	: TOF  			; // Timer off for internal axis enable 
	// Parameter read status 
		Cmd_EnDriveParRead	: BOOL 			; // Enable parameter read 
	// ===== Physical Homing signal =====
		IAxisHome AT %I* 	: BOOL 			; // Axis homing sensor from PLC (if MC_DefaultHoming is used)
END_VAR
VAR	// =============== Motion status functions ================
		fbMcReadAxisStatus	: MC_ReadStatus ;	// Fb for reading axis status	
	// =============== Motion function blocks =================
		fbMcPower 			: MC_Power		;		// FB for enable and override
		fbMcReset 			: MC_Reset		;		// FB to reset axis
		fbSoeReset			: FB_SoEReset	; 		// FB to reset axis hardware
		fbMcHome			: MC_Home		;		// Fb to home Axis
		fbMcStop 			: MC_Stop		;		// FB to stop axis
		fbMcHalt			: MC_Halt		;		// FB to halt axis
		fbMcJog				: MC_Jog		;		// FB to Jog axis
		fbMcMoveVelocity	: MC_MoveVelocity;		// FB to move with specified velocity until Next command is given
		fbMcGearInSlave		: MC_GearIn		;		// FB to gear axis to master 
		fbMcGearInDyn		: MC_GearInDyn	;		// FB to gear axis dynamicly to master
		fbMcGearOutSlave	: MC_GearOut	;		// FB to decouple gearing

	(* PtoP Motion move commands are in arrays so multiple commands can be stacked *) 
		fbMCMoveRelative	: ARRAY [0..1] OF MC_MoveRelative	;		// FB to move relative
		fbMcMoveAbsolute	: ARRAY [0..1] OF MC_MoveAbsolute	;		// FB to move axis (velocity movement)
		fbMcMoveModulo		: ARRAY [0..1] OF MC_MoveModulo		;		// FB to move axis to modulo position
	// ===== Safe commands =====
		bCmdSafeStop	: BOOL ;
		bCmdSafeSpeed	: BOOL ; 
	// ===== Function execute triggers =====
		bExec_Init 			: BOOL := FALSE; // Execute init 
		bExec_Reset			: BOOL := FALSE; // Execute reset
		bExec_Halt			: BOOL := FALSE; // Execute hold
		bExec_Home			: BOOL := FALSE; // Execute Home
		bExec_JogPositive	: BOOL := FALSE; // Execute Jog in positive direction
		bExec_JogNegative	: BOOL := FALSE; // Execute Jog in negative direction
		bExec_MoveVelocity	: BOOL := FALSE; // Execute move velocity
		bExec_Hardstop		: BOOL := FALSE; // Execute hardstop
		bExec_Softstop		: BOOL := FALSE; // Execute Softstop
		bExec_GearAsSlave	: BOOL := FALSE; // Execute gear as slave
		bExec_GearSlaveDyn	: BOOL := FALSE; // Execute gear slave dynamic
		bExec_GearOutSlave	: BOOL := FALSE; // execute gear out slave
	// ===== Move ristrictions ======
		bCmdLimitVelocity 	: BOOL := FALSE			; // velocity limiting is active 
		fCmdVelocityLimit	: LREAL:= fSafeVeloLimit; // Maximum velocity limit when velocity limiting is active  
	(* PtoP Motion move commands are in arrays so multiple commands can be stacked *) 
		arExec_MoveRelative	: ARRAY [0..1] OF BOOL ; // Execute move relative
		arExec_MoveAbs		: ARRAY [0..1] OF BOOL ; // Execute move absolute reverse
		arExec_MoveModulo	: ARRAY [0..1] OF BOOL ; // Execute move modulo
END_VAR
VAR
	// ===== Loop variables =====
		i : DINT := 0 ; // For loop increment
END_VAR

// ==== Check if axis is initiated =====
	IF NOT bInitDone THEN 
		RETURN ; 
	END_IF

// ===== Execute safe functions =====
	ExecSafeFunctions(); 

// ==== Execute organizational functions =====
	METH_ExecuteOrganizationFunctions();

// ==== execute motion functions =====
	METH_ExecuteMotionFunctions();

METHOD PUBLIC CmdGearDynamic : BOOL // Set axis to geared, activates with variable gear ratio until geared out or stopped (if method is no longer called then gear ratio is locked to last value)
VAR_INPUT
	fGearRatio	:	LREAL	:= 1	; // Slave Axis gearing ratio (Master = 1/ fGearRatio = Slave)	
END_VAR
// Set command to true 
bExec_GearSlaveDyn 	:= TRUE ;
bInternalEnable		:= TRUE ;

// coppy parameters
fCmdGearRatio 				:= fGearRatio ;

// Set feedback output 
CmdGearDynamic := fbMcGearInDyn.Active ;
END_METHOD

METHOD PUBLIC CmdGearIn : BOOL // Set axis to geared, activates with constant gear ratio until geared out or stopped
VAR_INPUT
	fGearRatio	:	LREAL	:= 1	; // Slave Axis gearing ratio (Master = 1/ fGearRatio = Slave)	
END_VAR
// Set command to true 
bExec_GearAsSlave 	:= TRUE ;
bInternalEnable		:= TRUE ;

// coppy parameters
fCmdGearRatio 				:= fGearRatio ;

// Set feedback output 
CmdGearIn := fbMcGearInSlave.Active ;
END_METHOD

METHOD CmdGearOut : BOOL
VAR_INPUT
END_VAR
// Set command to true
bExec_GearOutSlave := TRUE ;
bExec_GearSlaveDyn := FALSE;

// Set feedback Output
CmdGearOut := fbMcGearOutSlave.Done;
END_METHOD

METHOD PUBLIC CmdHalt : BOOL
VAR_INPUT
	fDeceleration 	: LREAL := 0 ; // command deceleration
	mcBuffermode	: MC_BufferMode ; // Buffermode defines how the previous command is executed.
END_VAR
// Set command to true 
bExec_Halt 		:= TRUE ;
bInternalEnable	:= TRUE ;

// coppy parameters
fbMcHalt.Deceleration	:= fDeceleration;
fbMcHalt.BufferMode		:= mcBuffermode	;

// Set feedback output 
CmdHalt := fbMchalt.Active ;
END_METHOD

METHOD PUBLIC CmdHome : BOOL // start axis homing procedure
VAR_INPUT
	fPosition 		: LREAL := 0 ; // Homing position
	mcBufferMode	: MC_BufferMode := MC_BufferMode.MC_Aborting		; // Buffermode
END_VAR
// set command to true 
bExec_Home 		:= TRUE	; 
bInternalEnable	:= TRUE ;

// coppy parameters
fbMcHome.Position 	:= fPosition 	;
fbMcHome.BufferMode	:= mcBufferMode ;

// Set feedback output
CmdHome := fbMcHome.Done ;
END_METHOD

METHOD PUBLIC CmdJog : BOOL // Jog axis with variable speed. jog stops as soon as the command is false
VAR_INPUT
	fVelocity		: LREAL 	; // jog velocity can be adjusted as long as the command is active
	fPos			: LREAL 	; // Jog position or step size (if aplicable)
	bJogNegative 	: BOOL 		:= FALSE ; // jog in negative direction
	eJogmode		: E_JogMode := E_JogMode.MC_JOGMODE_CONTINOUS ; // jogmode [default MC_JOGMODE_CONTINOUS] 
END_VAR
// Velocity conversion from RPM to deg/sec
	IF bIcfCmdVelocityRpm THEN 
		fVelocity := Rpm_To_DegS(fVelocity);
	END_IF

// Set command to true
	IF fbMcJog.Velocity = fVelocity THEN // If command velocity changes, then set exec to false for one cycle to trigger new velocity so the jog follows the set velocity
		bExec_JogPositive	:= NOT bJogNegative ;
		bExec_JogNegative 	:= bJogNegative ;
	END_IF
	bInternalEnable			:= TRUE ;

// coppy parameters
	fbMcJog.Velocity	:= fVelocity 	;
	fbmcjog.Mode		:= eJogmode		;
	fbMcJog.Position	:= fPos			;

// Set feedback output 
	CmdJog := fbMcJog.Active ;
END_METHOD

METHOD PUBLIC CmdLimitVelocity : BOOL // limit axis maximum velocity, stays active as long as command is called. 
VAR_INPUT
	fVelocityLimit	: LREAL ; // velocity Maximum limit
END_VAR
// Set velocity limiting command 
bCmdLimitVelocity S= TRUE;
	
// Set velocity maximum value 
fCmdVelocityLimit := fVelocityLimit ; 

// set feedback 
CmdLimitVelocity := bVelocityLimited ;
END_METHOD

METHOD PUBLIC CmdMoveAbs : BOOL // Move absolute command
VAR_INPUT
	fPosition	:	LREAL 	; // target position
	fVelocity	: 	LREAL 	; // Maximum velocity [units/sec]
	mcBuffermode: 	MC_BufferMode ; // Buffermode defines how the previous command is executed.
END_VAR
// Velocity conversion from RPM to deg/sec
	IF bIcfCmdVelocityRpm THEN 
		fVelocity := Rpm_To_DegS(fVelocity);
	END_IF

// Determine function for command stacking
	IF fbMcMoveAbsolute[0].Active THEN 
		arExec_MoveAbs[1] 				:= (fPosition <> fbMcMoveAbsolute[0].Position OR fVelocity <> fbMcMoveAbsolute[0].Velocity) ;
		fbMcMoveAbsolute[1].Position 	:= fPosition ;
		fbMcMoveAbsolute[1].Velocity 	:= fVelocity ; 
		fbMcMoveAbsolute[1].BufferMode 	:= mcBuffermode ;
	ELSE
		arExec_MoveAbs[0] 				:= (fPosition <> fbMcMoveAbsolute[1].Position OR fVelocity <> fbMcMoveAbsolute[1].Velocity) ;
		fbMcMoveAbsolute[0].Position 	:= fPosition ;
		fbMcMoveAbsolute[0].Velocity 	:= fVelocity ; 
		fbMcMoveAbsolute[0].BufferMode 	:= mcBuffermode ;
	END_IF

bInternalEnable	:= TRUE ;

(* // Reset position position and velocity commands
	IF fbMcMoveAbsolute[1].Active AND NOT fbMcMoveAbsolute[0].Busy THEN 
		fbMcMoveAbsolute[0].Velocity := 0 ;
		fbMcMoveAbsolute[0].Position := 0 ;
	ELSIF fbMcMoveAbsolute[0].Active AND NOT fbMcMoveAbsolute[1].Busy THEN 
		fbMcMoveAbsolute[1].Velocity := 0 ;
		fbMcMoveAbsolute[1].Position := 0 ;
 	END_IF 
*)
// set feedback
IF arExec_MoveAbs[1] OR fbMcMoveAbsolute[1].Busy THEN 
	CmdMoveAbs :=	fbMcMoveAbsolute[1].Active ;
ELSE 
	CmdMoveAbs :=	fbMcMoveAbsolute[0].Active ;
END_IF
END_METHOD

METHOD PUBLIC CmdMoveModulo : BOOL // Move to a modulo position
VAR_INPUT
	fPosition	:	LREAL 	; // target position
	fVelocity	: 	LREAL 	; // Maximum velocity [units/sec]
	mcDirection : 	MC_Direction := MC_Direction.MC_Positive_Direction ; // Direction of movement mc_direction [ deafult mc_positive_direction]
	mcBuffermode: 	MC_BufferMode ; // Buffermode defines how the previous command is executed.
END_VAR
// Velocity conversion from RPM to deg/sec
	IF bIcfCmdVelocityRpm THEN 
		fVelocity := Rpm_To_DegS(fVelocity);
	END_IF

// Determine function for command stacking
	IF fbMcMoveModulo[0].Active THEN 
		arExec_MoveModulo[1] 		:= (fPosition <> fbMcMoveModulo[0].Position OR fVelocity <> fbMcMoveModulo[0].Velocity)	;
		fbMcMoveModulo[1].Velocity 	:= fVelocity 	;
		fbMcMoveModulo[1].Position 	:= fPosition 	;
		fbMcMoveModulo[1].Direction	:= mcDirection	;
		fbMcMoveModulo[1].BufferMode:= mcBuffermode ;
	ELSE    
		arExec_MoveModulo[0] 		:= (fPosition <> fbMcMoveModulo[1].Position OR fVelocity <> fbMcMoveModulo[1].Velocity) ;
		fbMcMoveModulo[0].Velocity 	:= fVelocity 	;
		fbMcMoveModulo[0].Position 	:= fPosition 	;
		fbMcMoveModulo[0].Direction	:= mcDirection	;
		fbMcMoveModulo[0].BufferMode:= mcBuffermode ;
	END_IF

bInternalEnable	:= TRUE ;

(*// Reset position position and velocity commands
	IF fbMcMoveModulo[1].Active AND NOT fbMcMoveModulo[0].Busy THEN 
		fbMcMoveModulo[0].Velocity := 0 ;
		fbMcMoveModulo[0].Position := 0 ;
	ELSIF fbMcMoveModulo[0].Active AND NOT fbMcMoveModulo[1].Busy THEN 
		fbMcMoveModulo[1].Velocity := 0 ;
		fbMcMoveModulo[1].Position := 0 ;
 	END_IF 
*)
// set feedback
IF arExec_MoveModulo[1] OR fbMcMoveModulo[1].Busy THEN 
	CmdMoveModulo :=	fbMcMoveModulo[1].Active OR fbMcMoveModulo[1].Done;
ELSE
	CmdMoveModulo :=	fbMcMoveModulo[0].Active OR fbMcMoveModulo[0].Done ;
END_IF
END_METHOD

METHOD CmdMoveRelative : BOOL // move relative command 
VAR_INPUT
	fDistance	:	LREAL 	; // target position
	fVelocity	: 	LREAL 	; // Maximum velocity [units/sec]
	mcBuffermode: 	MC_BufferMode ; // Buffermode defines how the previous command is executed.
END_VAR
// Velocity conversion from RPM to deg/sec
	IF bIcfCmdVelocityRpm THEN 
		fVelocity := Rpm_To_DegS(fVelocity);
	END_IF

// Determine function for command stacking
	IF fbMCMoveRelative[0].Active THEN 
		arExec_MoveRelative[1] := (fDistance <> fbMCMoveRelative[0].Distance OR fVelocity <> fbMCMoveRelative[0].Velocity) ;
		fbMCMoveRelative[1].Velocity	:= fVelocity 	;
		fbMCMoveRelative[1].Distance	:= fDistance	;
		fbMCMoveRelative[1].BufferMode	:= mcBuffermode	;
	ELSE 
		arExec_MoveRelative[0] := (fDistance <> fbMCMoveRelative[1].Distance OR fVelocity <> fbMCMoveRelative[1].Velocity) ;
		fbMCMoveRelative[0].Velocity	:= fVelocity 	;
		fbMCMoveRelative[0].Distance	:= fDistance	;
		fbMCMoveRelative[0].BufferMode	:= mcBuffermode	;
	END_IF

bInternalEnable	:= TRUE ;

(*// Reset position position and velocity commands
	IF fbMCMoveRelative[1].Active AND NOT fbMCMoveRelative[0].Busy THEN 
		fbMCMoveRelative[0].Velocity := 0 ;
		fbMCMoveRelative[0].Distance := 0 ;
	ELSIF fbMCMoveRelative[0].Active AND NOT fbMCMoveRelative[1].Busy THEN 
		fbMCMoveRelative[1].Velocity := 0 ;
		fbMCMoveRelative[1].Distance := 0 ;
 	END_IF 
*)
// set feedback
IF arExec_MoveRelative[1] OR fbMCMoveRelative[1].Busy THEN 
	CmdMoveRelative :=	fbMCMoveRelative[1].Active ;
ELSE
	CmdMoveRelative :=	fbMCMoveRelative[0].Active ;
END_IF
END_METHOD

METHOD PUBLIC CmdMoveVelocity : BOOL // Move with set velocity until stopped
VAR_INPUT
	fVelocity	: 	LREAL 	; // Maximum velocity [units/sec]
	mcDirection : 	MC_Direction := MC_Direction.MC_Positive_Direction ; // Direction of movement mc_direction [ deafult mc_positive_direction]
	mcBuffermode: 	MC_BufferMode ; // Buffermode defines how the previous command is executed.
END_VAR
// Velocity conversion from RPM to deg/sec
	IF bIcfCmdVelocityRpm THEN 
		fVelocity := Rpm_To_DegS(fVelocity);
	END_IF

// Set command to true 
	bExec_MoveVelocity 	:= TRUE ;
	bInternalEnable		:= TRUE ;

// coppy parameters
	fbMcMoveVelocity.Velocity	:= fVelocity 	;
	fbMcMoveVelocity.Direction 	:= mcDirection	;
	fbMcMoveVelocity.BufferMode	:= mcBuffermode	;

// Set feedback output 
	CmdMoveVelocity := fbMcMoveVelocity.Active ;
END_METHOD

METHOD PUBLIC CmdReset : BOOL
VAR_INPUT
END_VAR
// Set reset axis to true 				
	bExec_Reset 	:= TRUE ; 
	bInternalEnable	:= TRUE ;
	
// Set feedback output 
	CmdReset := fbMcReset.Done ;
END_METHOD

METHOD PUBLIC CmdSafeSpeed : BOOL
VAR_INPUT
END_VAR
// Set safestop command
bCmdSafeSpeed := TRUE ; 

// Set feedback output 
CmdSafeSpeed := AxisRef.NcToPlc.ActVelo <= fSafeVeloLimit ;
END_METHOD

METHOD PUBLIC CmdSafeStop : BOOL
VAR_INPUT
END_VAR
// Set safestop command
bCmdSafeStop := TRUE ; 

// Set feedback output 
CmdSafeStop := bDevIsSafe ;
END_METHOD

METHOD PUBLIC Init : BOOL
VAR_INPUT
	// Axis message Data 
	sName	: STRING 	; // Name of the axis (used for fault handling and identification)
	sNumber	: UDINT		; // Axis number 
	// Config Bits
	bIcfCmdVelocityRpm	: BOOL ; // input speeds in Rpm
	bIcfEnableForward 	: BOOL ; // Enable forward motion
	bIcfEnablereverse	: BOOL ; // Enable reverse motion
	bIcfAlwaysEnable	: BOOL ; // 1 = Axis always enabled, 0 = Axis disabled at Idle 
	
